# B&R Automation Studio project NAEUL004C00R13L518F00 (part 46)

```iecst
END_ACTION
```

#### Act_OutputConfig.st
```iecst
ACTION Act_OutputConfig:
	// Output: Assign To Global For Independent Package Usage

	g_tyPshrConv := tylocalPshrConv.Out; // Change the Global Naming According to the Physical Hardware Module

END_ACTION
```

#### Cyclic.st
```iecst
(** 2019-03-29 **)
PROGRAM _CYCLIC

	IF bInitialDone = FALSE THEN
		IF g_tyStartUp.bNtSettingsLoadDone = TRUE  THEN
			bInitialDone	:= TRUE;
			Act_Initial;
		END_IF
	ELSE
		Act_InputConfig;
		IF (tylocalPshrConv.In.bPrep = TRUE) AND (tylocalPshrConv.In.bEn = TRUE) AND (tylocalPshrConv.In.bDis = FALSE) THEN
			Act_Link;
			Act_Main;
		ELSE
			IF tylocalPshrConv.Out.eStat <> ConvActIdle THEN
				tylocalPshrConv.Out.eStatus	:= Done;
			ELSE
				tylocalPshrConv.Out.eStatus	:= Idle;
			END_IF
		END_IF
		Act_OutputConfig;
		Act_Alarm;

	END_IF

END_PROGRAM
```

#### Init.st
```iecst
(** 2019-03-25 **)
PROGRAM _INIT

	(* Always Change If Project Change *)

	//Physical Configuration
	diInitTm	:= 0;

	//Pass Address To Global Address For External Use
	//Action, State & Status
	p_PshrConvStat		:= ADR(eStat);
	p_PshrConvStatus	:= ADR(eStatus);
	p_PshrConvStatTxt	:= ADR(sStatTxt);

	//Alarm
	p_PshrConvAlmData	:= ADR(tyAlmData);

	//Output
	p_PshrConvHvBrd						:= ADR(bHvBrd);
	p_PshrConvRejHvBrd					:= ADR(bRejHvBrd);
	p_PshrConvInspHvBrd					:= ADR(bInspHvBrd);
	p_PshrConvGdBrd						:= ADR(bGdBrd);
	p_PshrConvLmtSenActivated			:= ADR(bLmtSenActivated);
	p_PshrConvMtrSigOnOrLToR			:= ADR(bMtrSigOnOrLToR);
	p_PshrConvMtrDirOrRToL				:= ADR(bMtrDirOrRToL);

	p_PshrConvPshrExtCtrl				:= ADR(bPshrExtCtrl);
	p_PshrConvPshrRetCtrl				:= ADR(bPshrRetCtrl);
	p_PshrConvPshrTwoOutputControl		:= ADR(bPshrTwoOutputControl);
	p_PshrConvPshrExtended				:= ADR(bPshrExtended);
	p_PshrConvPshrRetracted				:= ADR(bPshrRetracted);

	p_PshrConvPullerExtCtrl				:= ADR(bPullerExtCtrl);
	p_PshrConvPullerRetCtrl				:= ADR(bPullerRetCtrl);
	p_PshrConvPullerTwoOutputControl	:= ADR(bPullerTwoOutputControl);
	p_PshrConvPullerExtended			:= ADR(bPullerExtended);
	p_PshrConvPullerRetracted			:= ADR(bPullerRetracted);

	p_PshrConvRotRemoteCtrl				:= ADR(bRotRemoteCtrl);
	p_PshrConvRotTwoOutputControl		:= ADR(bRotTwoOutputControl);
	p_PshrConvRotAtRemote				:= ADR(bRotAtRemote);
	p_PshrConvRotAtHome					:= ADR(bRotAtHome);

	p_PshrConvRejectUpCtrl				:= ADR(bRejectUpCtrl);
	p_PshrConvRejectDownCtrl			:= ADR(bRejectDownCtrl);
	p_PshrConvRejectTwoOutputControl	:= ADR(bRejectTwoOutputControl);
	p_PshrConvRejectAtUp				:= ADR(bRejectAtUp);
	p_PshrConvRejectAtDown				:= ADR(bRejectAtDown);
	//ADDED

	p_PshrConvPshrRetAllwTrav			:= ADR(bPshrRetAllwTraverse);

	(* Always Change If Project Change *)

END_PROGRAM
```

### MtrPshr.typ - Change By Project
```iecst
(*2019-06-17*)
(**)
(*Action*)

TYPE
	eMtrPshrAction :
		(
		MtrPshrActIdle,
		MtrPshrActExt,
		MtrPshrActRet,
		MtrPshrActStop,
		MtrPshrActSetExt,
		MtrPshrActRstExt,
		MtrPshrActSetRet,
		MtrPshrActRstRet,
		MtrPshrActSetSpdBit0,
		MtrPshrActRstSpdBit0,
		MtrPshrActSetSpdBit1,
		MtrPshrActRstSpdBit1,
		MtrPshrActSetSpdBit2,
		MtrPshrActRstSpdBit2,
		MtrPshrActSetSigOn,
		MtrPshrActRstSigOn,
		MtrPshrActSetBrake,
		MtrPshrActRstBrake,
		MtrPshrActSetAlmRst,
		MtrPshrActRstAlmRst,
		MtrPshrActSetAll,
		MtrPshrActRstAll
		);
	tyMtrPshr : 	STRUCT
		In : tyMtrPshrIn1;
		Out : tyMtrPshrOut1;
	END_STRUCT;
	tyMtrPshrIn1 : 	STRUCT
		eAct : eConvAction;
		udiRstErr : UDINT;
		bPrep : BOOL;
		bEn : BOOL;
		bDis : BOOL;
		bManual : BOOL;
		bDir : BOOL := FALSE;
		tAlmRstTm : TIME := T#1s;
		tAlmTrigTm : TIME := T#1s;
		tMtrBrkOffDlyTm : TIME := T#500ms;
		tExtTO : TIME := T#20s;
		tRetTO : TIME := T#20s;
		diExtSlowSpd : DINT;
		diRetSlowSpd : DINT;
		diExtNomSpd : {REDUND_UNREPLICABLE} DINT;
		diRetNomSpd : {REDUND_UNREPLICABLE} DINT;
		diExtTorque : DINT;
		diRetTorque : DINT;
		diStartTorque : DINT;
		bExtSen : BOOL;
		bRetSen : BOOL;
		bExtSlowSen : BOOL;
		bRetSlowSen : BOOL;
		bExtSafetySen : BOOL := TRUE;
		bRetSafetySen : BOOL := TRUE;
		bAlarmSig : BOOL;
		bTorqueSig : BOOL;
		bNtParamAutoRcpPrep : BOOL;
		bMcParamAutoRcpDis : BOOL;
		bLinkDISafetyRlySig : BOOL;
		bLinkPshrExtCtrl : BOOL;
		bLinkPshrRetCtrl : BOOL;
		bLinkAlarmSig : BOOL;
		sProgNm : STRING[15];
	END_STRUCT;
	tyMtrPshrOut1 : 	STRUCT
		eStat : eMagConv2ClpAction;
		eStatus : eFBStatus;
		sStatTxt : STRING[200];
		tyAlmData : tyAlmDat;
		bExtended : BOOL;
		bRetracted : BOOL;
		bCW : BOOL;
		bCCW : BOOL;
		bSpdBinBit0 : BOOL;
		bSpdBinBit1 : BOOL;
		bSpdBinBit2 : BOOL;
		bSigOn : BOOL;
		bBrake : BOOL;
		bAlmRst : BOOL;
	END_STRUCT;
END_TYPE
```

### MtrPshr.var - Change By Project
```iecst
VAR
	g_tyMtrPshr : tyMtrPshrOut1;
END_VAR
```

### Program Logical/MtrPshr/MtrPshr (IEC) - 1.00.0 - NtConv v5.00.0 , NtPneu v5.00.0

#### InputRef.var
```iecst
(*2019-03-25*)
(**)
(*General*)
VAR
	p_eAct : REFERENCE TO eMtrPshrAction;
	p_udiRstErr : REFERENCE TO UDINT;
	p_bPrep : REFERENCE TO BOOL;
	p_bEn : REFERENCE TO BOOL;
	p_bDis : REFERENCE TO BOOL;
END_VAR
(**)
(*Configuration*)
VAR
	p_bManual : REFERENCE TO BOOL;
	p_bDir : REFERENCE TO BOOL;
	p_tAlmRstTm : REFERENCE TO TIME;
	p_tAlmTrigTm : REFERENCE TO TIME;
	p_tMtrBrkOffDlyTm : REFERENCE TO TIME;
	p_tExtTO : REFERENCE TO TIME;
	p_tRetTO : REFERENCE TO TIME;
	p_diExtSlowSpd : REFERENCE TO DINT;
	p_diRetSlowSpd : REFERENCE TO DINT;
	p_diExtNomSpd : REFERENCE TO DINT;
	p_diRetNomSpd : REFERENCE TO DINT;
	p_diExtTorque : REFERENCE TO DINT;
	p_diRetTorque : REFERENCE TO DINT;
	p_diStartTorque : REFERENCE TO DINT;
	p_sProgNm : REFERENCE TO STRING[15];
	p_bNtSettingsLoadDone : REFERENCE TO BOOL;
END_VAR
(**)
(*Input*)
VAR
	p_bExtSen : REFERENCE TO BOOL;
	p_bRetSen : REFERENCE TO BOOL;
	p_bExtSlowSen : REFERENCE TO BOOL;
	p_bRetSlowSen : REFERENCE TO BOOL;
	p_bExtSafetySen : REFERENCE TO BOOL;
	p_bRetSafetySen : REFERENCE TO BOOL;
	p_bAlarmSig : REFERENCE TO BOOL;
	p_bTorqueSig : REFERENCE TO BOOL;
	p_bNtParamAutoRcpPrep : REFERENCE TO BOOL;
	p_bMcParamAutoRcpDis : REFERENCE TO BOOL;
END_VAR
```

#### InputRef_Link.var
```iecst
(*2019-04-09*)
(**)
VAR
	p_bLinkOpsRun : REFERENCE TO BOOL;
END_VAR
(**)
VAR
	p_bLinkDISafetyRlySig : REFERENCE TO BOOL;
	p_bLinkPshrExtCtrl : REFERENCE TO BOOL;
	p_bLinkPshrRetCtrl : REFERENCE TO BOOL;
	p_bLinkAlarmSig : REFERENCE TO BOOL;
END_VAR
```

#### Local.var
```iecst
(*2019-06-17*)
VAR
	tylocalMtrPshr : tyMtrPshr;
END_VAR
(**)
(*Local Action, State & Status*)
VAR
	udiStatus : UDINT := 0;
	a_sStatText : ARRAY[0..60] OF STRING[200] := ['Idling','Extending','Retracting','Stopping','Turning On Motor Extend','Turning Off Motor Extend','Turning On Motor Retract','Turning Off Motor Retract','Turning On Speed Binary Bit 0','Turning Off Speed Binary Bit 0','Turning On Speed Binary Bit 1','Turning Off Speed Binary Bit 1','Turning On Speed Binary Bit 2','Turning Off Speed Binary Bit 2','Turning On Signal On','Turning Off Signal On','Turning On Brake','Turning Off Brake','Turning On Alarm Reset','Turning Off Alarm Reset','Turning On All Motor Output','Turning Of All Motor Output',39('')];
END_VAR
(**)
(*Local Alarm*)
VAR
	tyAlmData : tyAlmDat;
END_VAR
(**)
(*Local*)
VAR
	bRstErr : BOOL;
	udiRstErrOld : UDINT;
	bInitDone : BOOL;
	bInitialDone : BOOL;
	eStatOld : eMtrPshrAction := MtrPshrActIdle;
	iAnalogTorque : INT;
	diMtrSpd : DINT;
	bMtrSpdSlw : BOOL;
	fbAlmRstTm : TON := (PT:=T#1s);
	fbAlmTrigTm : TON := (PT:=T#2s);
	fbMtrBrkOffDlyTm : TON;
	fbMtrPshrExtChk : fbPneuExtRetSenExtChk;
	fbMtrPshrRetChk : fbPneuExtRetSenRetChk;
	udiModuleNum : UDINT := 2201;
END_VAR
```

#### Act_Action.st
```iecst
(** 2019-03-25 **)
ACTION Act_Action:

	//Reset Error
	IF (eStatus = Error) AND bRstErr THEN
		p_eAct	:= MtrPshrActIdle;
		eStat	:= MtrPshrActIdle;
	END_IF

	//Set p_eAct
	IF eStatus = Idle OR eStatus = Busy OR eStatus = Done THEN
		eStat	:= p_eAct;
	END_IF

END_ACTION
```

#### Act_Alarm.st
```iecst
(** 2019-03-25 **)
ACTION Act_Alarm:
	//Reset Error
	IF (tylocalMtrPshr.Out.eStatus = Error) AND bRstErr THEN
		tylocalMtrPshr.In.eAct	:= MtrPshrActIdle;
		tylocalMtrPshr.Out.eStat	:= MtrPshrActIdle;
	END_IF

	IF tylocalMtrPshr.In.udiRstErr <> udiRstErrOld THEN
		bRstErr			:= TRUE;
		udiRstErrOld	:= tylocalMtrPshr.In.udiRstErr;
	ELSE
		bRstErr			:= FALSE;
	END_IF
	//Error
	IF EDGEPOS(eStatus = Error) THEN

		tylocalMtrPshr.Out.tyAlmData.udiCode		:= udiStatus;
		tylocalMtrPshr.Out.tyAlmData.eSeverity		:= AlmSeverityError;
		tylocalMtrPshr.Out.tyAlmData.udiRunTime	:= tylocalMtrPshr.Out.tyAlmData.udiRunTime + 1;
		tylocalMtrPshr.Out.tyAlmData.bAlm			:= TRUE;
		tylocalMtrPshr.Out.tyAlmData.udiModuleNum  := udiModuleNum;
		g_tyAlmProgNm.sMtrPshrProgNm		    := tylocalMtrPshr.In.sProgNm;

		tylocalMtrPshr.Out.sStatTxt	:= tylocalMtrPshr.Out.tyAlmData.sAlmMsg;

	ELSIF bRstErr AND (tyAlmData.udiCode <> 0) THEN

		tylocalMtrPshr.Out.tyAlmData.udiCode	:= 0;
		tylocalMtrPshr.Out.tyAlmData.eSeverity	:= AlmSeverityNA;
		tylocalMtrPshr.Out.tyAlmData.bAlm			:= FALSE;
		tylocalMtrPshr.Out.sStatTxt	:= a_sStatText[tylocalMtrPshr.Out.eStat];

	END_IF

END_ACTION
```

#### Act_Background.st
```iecst
(** 2019-01-18 **)
ACTION Act_Background:

	//background
	IF tylocalMtrPshr.In.bExtSen = FALSE THEN
		tylocalMtrPshr.Out.bExtended	:= FALSE;
	END_IF

	IF tylocalMtrPshr.In.bRetSen = FALSE THEN
		tylocalMtrPshr.Out.bRetracted	:= FALSE;
	END_IF

	//Torque Minimum Value
	IF iAnalogTorque < 1500 THEN
		iAnalogTorque	:= 1500;
	END_IF

	//Abnormal Movement
	IF tylocalMtrPshr.Out.eStatus <> Error THEN

		fbAlmTrigTm(IN := NOT tylocalMtrPshr.In.bAlarmSig);

		IF fbAlmTrigTm.Q = TRUE THEN
			tylocalMtrPshr.Out.eStatus		:= Error;
			udiStatus	:= 10006;	//Motorized Pusher Alarm Occur

			tylocalMtrPshr.Out.bCW			:= FALSE;
			tylocalMtrPshr.Out.bCCW		:= FALSE;
			tylocalMtrPshr.Out.bSpdBinBit0	:= FALSE;
			tylocalMtrPshr.Out.bSpdBinBit1	:= FALSE;
			tylocalMtrPshr.Out.bSpdBinBit2	:= FALSE;
			tylocalMtrPshr.Out.bSigOn		:= FALSE;
			tylocalMtrPshr.Out.bBrake		:= FALSE;
			tylocalMtrPshr.Out.bAlmRst		:= FALSE;

			tylocalMtrPshr.In.eAct	:= MtrPshrActIdle;
			tylocalMtrPshr.Out.eStat	:= MtrPshrActIdle;
		END_IF

	END_IF

	//Reset Error
	IF (tylocalMtrPshr.Out.eStatus = Error) AND bRstErr THEN
		IF tylocalMtrPshr.In.bAlarmSig = FALSE THEN
			tylocalMtrPshr.Out.bAlmRst			:= TRUE;
			fbAlmRstTm.IN	:= TRUE;
			fbAlmTrigTm(IN := FALSE);
		END_IF
	END_IF

	fbAlmRstTm;

	IF fbAlmRstTm.Q = TRUE THEN
		tylocalMtrPshr.Out.bAlmRst		:= FALSE;
		tylocalMtrPshr.Out.eStatus		:= Idle;
		udiStatus	:= 0;

		fbAlmRstTm.IN	:= FALSE;
	END_IF
END_ACTION
```

#### Act_InitGlobal.st
```iecst
(** 2019-04-09 **)
ACTION Act_InitGlobal:

	(* Always Change If Project Change *)

	//Pass Data To Link
	p_bLinkOpsRun ACCESS p_OpsRun;

	p_bLinkDISafetyRlySig ACCESS p_DISafetyRlySig;
	p_bLinkPshrExtCtrl ACCESS p_PshrConvPshrExtCtrl;
	p_bLinkPshrRetCtrl ACCESS p_PshrConvPshrRetCtrl;
	p_bLinkAlarmSig ACCESS p_DIMtrPshrAlmSig;

	//Pass Data To Internal Use
	p_udiRstErr ACCESS p_RstErrReset;
	p_bPrep ACCESS p_NtParamProjMotorizedPusherPrep;
	p_bManual ACCESS p_UIMnlMod;
	p_bDir ACCESS p_NtParamMtrPshrDir;
	p_tExtTO ACCESS p_NtParamMtrPshrExtTO;
	p_tRetTO ACCESS p_NtParamMtrPshrRetTO;
	p_diExtSlowSpd ACCESS p_NtParamMtrPshrExtSlowSpd;
	p_diRetSlowSpd ACCESS p_NtParamMtrPshrRetSlowSpd;
	p_diRetNomSpd ACCESS p_NtParamMtrPshrRetNomSpd;
	p_diRetTorque ACCESS p_NtParamMtrPshrRetTorq;
	p_diStartTorque ACCESS p_NtParamMtrPshrStartTorq;
	p_sProgNm ACCESS p_NtParamMtrPshrProgNm;
	p_bNtSettingsLoadDone ACCESS p_StartupNtSettingsLoadDone;

	p_bExtSen ACCESS p_DIPusherExtRS;
	p_bRetSen ACCESS p_DIPusherRetRS;
	p_bExtSlowSen ACCESS p_DIPusherExtSlwSen;
	p_bRetSlowSen ACCESS p_DIPusherRetSlwSen;
//	p_bAlarmSig ACCESS p_DIMtrPshrAlmSig;
	p_bTorqueSig ACCESS p_DIMtrPshrTorqueSig;

	p_bNtParamAutoRcpPrep ACCESS p_NtParamAutoRcpPrep ;
	p_bMcParamAutoRcpDis  ACCESS p_McParamAutoRcpDisable;
	(* Always Change If Project Change *)

END_ACTION
```

#### Act_Initial.st
```iecst
(** 2019-03-22 **)
ACTION Act_Initial:

	//Initial
	tylocalMtrPshr.Out.sStatTxt	:=  a_sStatText[eStat];

	fbAlmRstTm(IN := FALSE);
	fbAlmTrigTm(IN := FALSE);
	fbMtrBrkOffDlyTm(IN :=FALSE);
	fbMtrPshrExtChk(bEn	:=FALSE);
	fbMtrPshrRetChk(bEn	:=FALSE);

END_ACTION
```

#### Act_InitLocal.st
```iecst
(** 2019-03-25 **)
ACTION Act_InitLocal:

	//Input Reference Link To Local Variable
	p_eAct ACCESS ADR(eAct);
	p_udiRstErr ACCESS ADR(udiRstErr);
	p_bPrep ACCESS ADR(bPrep);
	p_bEn ACCESS ADR(bEn);
	p_bDis ACCESS ADR(bDis);

	p_bManual ACCESS ADR(bManual);
	p_bDir ACCESS ADR(bDir);
	p_tAlmRstTm ACCESS ADR(tAlmRstTm);
	p_tAlmTrigTm ACCESS ADR(tAlmTrigTm);
	p_tMtrBrkOffDlyTm ACCESS ADR(tMtrBrkOffDlyTm);
	p_tExtTO ACCESS ADR(tExtTO);
	p_tRetTO ACCESS ADR(tRetTO);
	p_diExtSlowSpd ACCESS ADR(diExtSlowSpd);
	p_diRetSlowSpd ACCESS ADR(diRetSlowSpd);
	p_diExtNomSpd ACCESS ADR(diExtNomSpd);
	p_diRetNomSpd ACCESS ADR(diRetNomSpd);
	p_diExtTorque ACCESS ADR(diExtTorque);
	p_diRetTorque ACCESS ADR(diRetTorque);
	p_diStartTorque ACCESS ADR(diStartTorque);
	p_sProgNm ACCESS ADR(sProgNm);
	p_bNtSettingsLoadDone ACCESS ADR(bNtSettingsLoadDone);

	p_bExtSen ACCESS ADR(bExtSen);
	p_bRetSen ACCESS ADR(bRetSen);
	p_bExtSlowSen ACCESS ADR(bExtSlowSen);
	p_bRetSlowSen ACCESS ADR(bRetSlowSen);
	p_bExtSafetySen ACCESS ADR(bExtSafetySen);
	p_bRetSafetySen ACCESS ADR(bRetSafetySen);
	p_bAlarmSig ACCESS ADR(bAlarmSig);
	p_bTorqueSig ACCESS ADR(bTorqueSig);

END_ACTION
```

#### Act_InputConfig.st
```iecst
(** 2019-04-09 **)
ACTION Act_InputConfig:

	(* Always Change If Project Change *)

	//Pass Data To Link

	tylocalMtrPshr.In.bLinkDISafetyRlySig := g_tyDISafetyRlySig;
	tylocalMtrPshr.In.bLinkPshrExtCtrl := g_tyPshrConvPshrExtCtrl;
	tylocalMtrPshr.In.bLinkPshrRetCtrl := g_tyPshrConvPshrRetCtrl;
	tylocalMtrPshr.In.bLinkAlarmSig := g_tyDIMtrPshrAlmSig;

	//Pass Data To Internal Use
	tylocalMtrPshr.In.udiRstErr := g_tyRstErrReset;
	tylocalMtrPshr.In.bPrep := g_tyNtParamProjMotorizedPusherPrep;
	tylocalMtrPshr.In.bManual := g_tyUIMnlMod;
	tylocalMtrPshr.In.bDir := g_tyNtParamMtrPshrDir;
	tylocalMtrPshr.In.tExtTO := g_tyNtParamMtrPshrExtTO;
	tylocalMtrPshr.In.tRetTO := g_tyNtParamMtrPshrRetTO;
	tylocalMtrPshr.In.diExtSlowSpd := g_tyNtParamMtrPshrExtSlowSpd;
	tylocalMtrPshr.In.diRetSlowSpd := g_tyNtParamMtrPshrRetSlowSpd;
	tylocalMtrPshr.In.diRetNomSpd := g_tyNtParamMtrPshrRetNomSpd;
	tylocalMtrPshr.In.diRetTorque := g_tyNtParamMtrPshrRetTorq;
	tylocalMtrPshr.In.diStartTorque := g_tyNtParamMtrPshrStartTorq;
	tylocalMtrPshr.In.sProgNm := g_tyNtParamCurr.sMtrPshrProgNm;

	tylocalMtrPshr.In.bExtSen := g_tyDIPusherExtRS;
	tylocalMtrPshr.In.bRetSen := g_tyDIPusherRetRS;
	tylocalMtrPshr.In.bExtSlowSen := g_tyDIPusherExtSlwSen;
	tylocalMtrPshr.In.bRetSlowSen := g_tyDIPusherRetSlwSen;
//	tylocalMtrPshr.In.bAlarmSig := g_tyDIMtrPshrAlmSig;
	tylocalMtrPshr.In.bTorqueSig := g_tyDIMtrPshrTorqueSig;

	tylocalMtrPshr.In.bNtParamAutoRcpPrep := g_tyNtParamAutoRcpPrep ;
	tylocalMtrPshr.In.bMcParamAutoRcpDis  := g_tyMcParamAutoRcpDisable;
	(* Always Change If Project Change *)

	IF g_tyOps.bRun THEN

		IF (tylocalMtrPshr.Out.eStatus <> Busy AND tylocalMtrPshr.Out.eStatus <> Idle)OR (tylocalMtrPshr.In.bLinkPshrExtCtrl = FALSE AND tylocalMtrPshr.In.bLinkPshrRetCtrl = FALSE)  THEN
			tylocalMtrPshr.In.eAct := MtrPshrActIdle;
		ELSIF tylocalMtrPshr.In.bLinkPshrExtCtrl AND tylocalMtrPshr.In.bLinkPshrRetCtrl = FALSE
			AND tylocalMtrPshr.In.bExtSen = FALSE
			THEN
			tylocalMtrPshr.In.eAct := MtrPshrActExt;

		ELSIF tylocalMtrPshr.In.bLinkPshrExtCtrl = FALSE AND tylocalMtrPshr.In.bLinkPshrRetCtrl
			AND tylocalMtrPshr.In.bRetSen = FALSE
			THEN
			tylocalMtrPshr.In.eAct := MtrPshrActRet;
		END_IF

	ELSIF tylocalMtrPshr.In.bManual = TRUE THEN

		IF (tylocalMtrPshr.Out.eStatus <> Busy AND tylocalMtrPshr.Out.eStatus <> Idle)OR (tylocalMtrPshr.In.bLinkPshrExtCtrl = FALSE AND tylocalMtrPshr.In.bLinkPshrRetCtrl = FALSE)  THEN
			tylocalMtrPshr.In.eAct := MtrPshrActIdle;
		ELSIF tylocalMtrPshr.In.bLinkPshrExtCtrl AND tylocalMtrPshr.In.bLinkPshrRetCtrl = FALSE
			AND tylocalMtrPshr.In.bExtSen = FALSE
			THEN
			tylocalMtrPshr.In.eAct := MtrPshrActExt;

		ELSIF tylocalMtrPshr.In.bLinkPshrExtCtrl = FALSE AND tylocalMtrPshr.In.bLinkPshrRetCtrl
			AND tylocalMtrPshr.In.bRetSen = FALSE
			THEN
			tylocalMtrPshr.In.eAct := MtrPshrActRet;
		END_IF

	ELSE
		tylocalMtrPshr.In.eAct := MtrPshrActIdle;
	END_IF
END_ACTION
```

#### Act_Link.st
```iecst
(** 2019-03-29 **)
ACTION Act_Link:

	IF tylocalMtrPshr.In.bLinkDISafetyRlySig = FALSE THEN
		tylocalMtrPshr.Out.bExtended	:= FALSE;
		tylocalMtrPshr.Out.bRetracted	:= FALSE;
	END_IF

	IF tylocalMtrPshr.In.bManual = TRUE THEN
		tylocalMtrPshr.In.diExtNomSpd ACCESS ADR(g_tyUIMnlMtrPshrExtSpd);
		tylocalMtrPshr.In.diExtTorque ACCESS ADR(g_tyUIMnlMtrPshrExtTorq);
	ELSE
		IF tylocalMtrPshr.In.bNtParamAutoRcpPrep AND NOT(tylocalMtrPshr.In.bMcParamAutoRcpDis) THEN
			tylocalMtrPshr.In.diExtNomSpd ACCESS g_tyProdRcpCurrRcp0MtrPshrExtSpd;
			tylocalMtrPshr.In.diExtTorque ACCESS g_tyProdRcpCurrRcp0MtrPshrExtTorq;
		ELSE
			tylocalMtrPshr.In.diExtNomSpd ACCESS  g_tyProdRcpCurrRcp1MtrPshrExtSpd;
			tylocalMtrPshr.In.diExtTorque ACCESS g_tyProdRcpCurrRcp1MtrPshrExtTorq;
		END_IF
	END_IF

	IF tylocalMtrPshr.In.bLinkDISafetyRlySig = TRUE THEN
		tylocalMtrPshr.In.bAlarmSig := tylocalMtrPshr.In.bLinkAlarmSig;
	ELSE
		tylocalMtrPshr.In.bAlarmSig := TRUE;
	END_IF

END_ACTION
```

#### Act_LinkAction.st
```iecst
(** 2019-04-09 **)
ACTION Act_LinkAction:

	IF p_bLinkOpsRun = TRUE THEN
		//	p_eAct ACCESS p_OpsTravULMtrPshrAct;
		IF p_bLinkPshrExtCtrl AND p_bLinkPshrRetCtrl = FALSE
			AND p_bExtSen = FALSE
			THEN
				p_eAct := MtrPshrActExt;

		ELSIF p_bLinkPshrExtCtrl = FALSE AND p_bLinkPshrRetCtrl
			AND p_bRetSen = FALSE
			THEN
				p_eAct := MtrPshrActRet;

		ELSE
				p_eAct := MtrPshrActIdle;
		END_IF

	ELSIF p_bManual = TRUE THEN
//		IF p_UIMtrPshrAct = MtrPshrActStop THEN
//			p_eAct := MtrPshrActStop;
//		ELSE
			IF p_bLinkPshrExtCtrl AND p_bLinkPshrRetCtrl = FALSE
			AND p_bExtSen = FALSE
				THEN
				p_eAct := MtrPshrActExt;

			ELSIF p_bLinkPshrExtCtrl = FALSE AND p_bLinkPshrRetCtrl
				AND p_bRetSen = FALSE
				THEN
				p_eAct := MtrPshrActRet;

			ELSE
				p_eAct := MtrPshrActIdle;
			END_IF
//		END_IF

	ELSE
			p_eAct := MtrPshrActIdle;
	END_IF

END_ACTION
```

#### Act_LinkEn.st
```iecst
(** 2019-01-11 **)
ACTION Act_LinkEn:

	//Link bPrep, bEn & bDis
	//p_bEn	:= FALSE;

END_ACTION
```

#### Act_Main.st
```iecst
(** 2019-06-17 **)
ACTION Act_Main:

	fbAlmRstTm.PT				:= tylocalMtrPshr.In.tAlmRstTm;
	fbAlmTrigTm.PT				:= tylocalMtrPshr.In.tAlmTrigTm;
	fbMtrBrkOffDlyTm.PT			:= tylocalMtrPshr.In.tMtrBrkOffDlyTm;
	fbMtrPshrExtChk.tTimeOut	:= tylocalMtrPshr.In.tExtTO;
	fbMtrPshrRetChk.tTimeOut	:= tylocalMtrPshr.In.tRetTO;
	//Set tylocalMtrPshr.In.eAct
	IF tylocalMtrPshr.Out.eStatus = Idle OR tylocalMtrPshr.Out.eStatus = Busy OR tylocalMtrPshr.Out.eStatus = Done THEN
		tylocalMtrPshr.Out.eStat	:= tylocalMtrPshr.In.eAct;
	END_IF

	IF eStatOld <> tylocalMtrPshr.Out.eStat THEN
		bMtrSpdSlw	:= FALSE;

		fbMtrBrkOffDlyTm(IN := FALSE);
		fbMtrPshrExtChk(bEn := FALSE);
		fbMtrPshrRetChk(bEn := FALSE);

		IF eStatOld <> MtrPshrActIdle
			AND eStatOld <> MtrPshrActSetExt
			AND eStatOld <> MtrPshrActRstExt
			AND eStatOld <> MtrPshrActSetRet
			AND eStatOld <> MtrPshrActRstRet
			AND eStatOld <> MtrPshrActSetSpdBit0
			AND eStatOld <> MtrPshrActRstSpdBit0
			AND eStatOld <> MtrPshrActSetSpdBit1
			AND eStatOld <> MtrPshrActRstSpdBit1
			AND eStatOld <> MtrPshrActSetSpdBit2
			AND eStatOld <> MtrPshrActRstSpdBit2
			AND eStatOld <> MtrPshrActSetSigOn
			AND eStatOld <> MtrPshrActRstSigOn
			AND eStatOld <> MtrPshrActSetBrake
			AND eStatOld <> MtrPshrActRstBrake
			AND eStatOld <> MtrPshrActSetAlmRst
			AND eStatOld <> MtrPshrActRstAlmRst
			AND eStatOld <> MtrPshrActSetAll
			AND eStatOld <> MtrPshrActRstAll THEN

			tylocalMtrPshr.Out.bCW			:= FALSE;
			tylocalMtrPshr.Out.bCCW		:= FALSE;
			tylocalMtrPshr.Out.bSpdBinBit0	:= FALSE;
			tylocalMtrPshr.Out.bSpdBinBit1	:= FALSE;
			tylocalMtrPshr.Out.bSpdBinBit2	:= FALSE;
			tylocalMtrPshr.Out.bSigOn		:= FALSE;
			tylocalMtrPshr.Out.bBrake		:= FALSE;
			tylocalMtrPshr.Out.bAlmRst		:= FALSE;

		END_IF

		sStatTxt	:= a_sStatText[tylocalMtrPshr.Out.eStat];

		eStatOld	:= tylocalMtrPshr.Out.eStat;

		tylocalMtrPshr.Out.eStatus		:= Busy;
	END_IF

	//Main
	CASE tylocalMtrPshr.Out.eStat OF

		MtrPshrActIdle:
			IF EDGENEG(tylocalMtrPshr.In.bManual) THEN
				tylocalMtrPshr.Out.bCW			:= FALSE;
				tylocalMtrPshr.Out.bCCW		:= FALSE;
				tylocalMtrPshr.Out.bSpdBinBit0	:= FALSE;
				tylocalMtrPshr.Out.bSpdBinBit1	:= FALSE;
				tylocalMtrPshr.Out.bSpdBinBit2	:= FALSE;
				tylocalMtrPshr.Out.bSigOn		:= FALSE;
				tylocalMtrPshr.Out.bBrake		:= FALSE;
				tylocalMtrPshr.Out.bAlmRst		:= FALSE;
			END_IF

			tylocalMtrPshr.Out.eStatus	:= Idle;

		MtrPshrActExt:
			IF tylocalMtrPshr.Out.eStatus = Idle OR tylocalMtrPshr.Out.eStatus = Busy THEN
				tylocalMtrPshr.Out.eStatus	:= Busy;

				//Motor Torque
				IF (tylocalMtrPshr.In.bRetSen OR tylocalMtrPshr.In.bRetSlowSen) THEN// OR  NOT(bMtrSpdSlw) THEN
					iAnalogTorque	:= ((DINT_TO_INT(tylocalMtrPshr.In.diStartTorque) * 16383) / 100); //5V at 16383 for maximum Torque
				ELSE //IF bMtrSpdSlw THEN
					iAnalogTorque	:= ((DINT_TO_INT(tylocalMtrPshr.In.diExtTorque) * 16383) / 100);
				END_IF

				IF iAnalogTorque < 1500 THEN
					iAnalogTorque	:= 1500;
				END_IF

				//Motor Speed
				IF tylocalMtrPshr.In.bExtSlowSen = TRUE OR tylocalMtrPshr.In.bTorqueSig = TRUE THEN
					bMtrSpdSlw	:= TRUE;
				END_IF

				IF bMtrSpdSlw = TRUE THEN
					diMtrSpd	:= tylocalMtrPshr.In.diExtSlowSpd;
				ELSE
					diMtrSpd	:= tylocalMtrPshr.In.diExtNomSpd;
				END_IF

				CASE diMtrSpd OF
					1:
						tylocalMtrPshr.Out.bSpdBinBit0	:= FALSE;
						tylocalMtrPshr.Out.bSpdBinBit1	:= FALSE;
						tylocalMtrPshr.Out.bSpdBinBit2	:= FALSE;
					2:
						tylocalMtrPshr.Out.bSpdBinBit0	:= TRUE;
						tylocalMtrPshr.Out.bSpdBinBit1	:= FALSE;
						tylocalMtrPshr.Out.bSpdBinBit2	:= FALSE;
					3:
						tylocalMtrPshr.Out.bSpdBinBit0	:= FALSE;
						tylocalMtrPshr.Out.bSpdBinBit1	:= TRUE;
						tylocalMtrPshr.Out.bSpdBinBit2	:= FALSE;
					4:
						tylocalMtrPshr.Out.bSpdBinBit0	:= TRUE;
						tylocalMtrPshr.Out.bSpdBinBit1	:= TRUE;
						tylocalMtrPshr.Out.bSpdBinBit2	:= FALSE;
					5:
						tylocalMtrPshr.Out.bSpdBinBit0	:= FALSE;
						tylocalMtrPshr.Out.bSpdBinBit1	:= FALSE;
						tylocalMtrPshr.Out.bSpdBinBit2	:= TRUE;
					6:
						tylocalMtrPshr.Out.bSpdBinBit0	:= TRUE;
						tylocalMtrPshr.Out.bSpdBinBit1	:= FALSE;
						tylocalMtrPshr.Out.bSpdBinBit2	:= TRUE;
					7:
						tylocalMtrPshr.Out.bSpdBinBit0	:= FALSE;
						tylocalMtrPshr.Out.bSpdBinBit1	:= TRUE;
						tylocalMtrPshr.Out.bSpdBinBit2	:= TRUE;
					8:
						tylocalMtrPshr.Out.bSpdBinBit0	:= TRUE;
						tylocalMtrPshr.Out.bSpdBinBit1	:= TRUE;
						tylocalMtrPshr.Out.bSpdBinBit2	:= TRUE;
				END_CASE

				//Motor On
				tylocalMtrPshr.Out.bSigOn	:= FALSE;
				tylocalMtrPshr.Out.bBrake	:= TRUE;

				IF tylocalMtrPshr.In.bDir = TRUE THEN
					tylocalMtrPshr.Out.bCW		:= TRUE;
				ELSE
					tylocalMtrPshr.Out.bCCW	:= TRUE;
				END_IF

				//Checking Extend
				fbMtrPshrExtChk.bExtSen		:= tylocalMtrPshr.In.bExtSen;
				fbMtrPshrExtChk.bRetSen		:= tylocalMtrPshr.In.bRetSen;
				fbMtrPshrExtChk.bExtSafety	:= tylocalMtrPshr.In.bExtSafetySen;

				fbMtrPshrExtChk(bEn := TRUE);

				IF fbMtrPshrExtChk.udiStatus = 0 THEN

					tylocalMtrPshr.Out.bSigOn	:= TRUE;
					tylocalMtrPshr.Out.bBrake	:= FALSE;
					tylocalMtrPshr.Out.bCW		:= FALSE;
					tylocalMtrPshr.Out.bCCW	:= FALSE;

					fbMtrBrkOffDlyTm(IN := TRUE);

					IF fbMtrBrkOffDlyTm.Q = TRUE THEN
						fbMtrBrkOffDlyTm(IN := FALSE);

						tylocalMtrPshr.Out.bCW			:= FALSE;
						tylocalMtrPshr.Out.bCCW		:= FALSE;
						tylocalMtrPshr.Out.bSpdBinBit0	:= FALSE;
						tylocalMtrPshr.Out.bSpdBinBit1	:= FALSE;
						tylocalMtrPshr.Out.bSpdBinBit2	:= FALSE;
						tylocalMtrPshr.Out.bSigOn		:= FALSE;
						tylocalMtrPshr.Out.bBrake		:= FALSE;

						tylocalMtrPshr.Out.bExtended	:= TRUE;
						tylocalMtrPshr.Out.eStatus		:= Done;
					END_IF

				ELSIF fbMtrPshrExtChk.udiStatus < 65534 THEN

					tylocalMtrPshr.Out.bCW			:= FALSE;
					tylocalMtrPshr.Out.bCCW		:= FALSE;
					tylocalMtrPshr.Out.bSpdBinBit0	:= FALSE;
					tylocalMtrPshr.Out.bSpdBinBit1	:= FALSE;
					tylocalMtrPshr.Out.bSpdBinBit2	:= FALSE;
					tylocalMtrPshr.Out.bSigOn		:= TRUE;
					tylocalMtrPshr.Out.bBrake		:= FALSE;

					tylocalMtrPshr.Out.bExtended	:= FALSE;
					tylocalMtrPshr.Out.eStatus		:= Error;

					IF fbMtrPshrExtChk.udiStatus = 1506 THEN
						udiStatus	:= 10000;	//Pusher Retract Sensor Off Time Out In Extend Check While Pusher Extend
					ELSIF fbMtrPshrExtChk.udiStatus = 1503 THEN
						udiStatus	:= 10001;	//Pusher Extend Sensor On Time Out In Extend Check While Pusher Extend
					ELSIF fbMtrPshrExtChk.udiStatus = 1507 THEN
						udiStatus	:= 10002;	//Pusher Extend Safety Sensor Error In Extend Check While Pusher Extend
					ELSE
						udiStatus	:= fbMtrPshrExtChk.udiStatus;
					END_IF

				END_IF

			END_IF

		MtrPshrActRet:
			IF tylocalMtrPshr.Out.eStatus = Idle OR tylocalMtrPshr.Out.eStatus = Busy THEN
				tylocalMtrPshr.Out.eStatus	:= Busy;

				//Motor Torque
				IF (tylocalMtrPshr.In.bExtSen OR tylocalMtrPshr.In.bExtSlowSen) THEN //OR NOT(bMtrSpdSlw) THEN
					iAnalogTorque	:= ((DINT_TO_INT(tylocalMtrPshr.In.diStartTorque) * 16383) / 100); //32767 ==10V ,10000 == 3v
				ELSE // bMtrSpdSlw THEN
					iAnalogTorque	:= ((DINT_TO_INT(tylocalMtrPshr.In.diRetTorque) * 16383) / 100);
				END_IF

				IF iAnalogTorque < 1500 THEN
					iAnalogTorque	:= 1500;
				END_IF

				//Motor Speed
				IF tylocalMtrPshr.In.bRetSlowSen = TRUE THEN
					bMtrSpdSlw	:= TRUE;
				END_IF

				IF bMtrSpdSlw = TRUE THEN
					diMtrSpd	:= tylocalMtrPshr.In.diRetSlowSpd;
				ELSE
					diMtrSpd	:= tylocalMtrPshr.In.diRetNomSpd;
				END_IF

				CASE diMtrSpd OF
					1:
						tylocalMtrPshr.Out.bSpdBinBit0	:= FALSE;
						tylocalMtrPshr.Out.bSpdBinBit1	:= FALSE;
						tylocalMtrPshr.Out.bSpdBinBit2	:= FALSE;
					2:
						tylocalMtrPshr.Out.bSpdBinBit0	:= TRUE;
						tylocalMtrPshr.Out.bSpdBinBit1	:= FALSE;
						tylocalMtrPshr.Out.bSpdBinBit2	:= FALSE;
					3:
						tylocalMtrPshr.Out.bSpdBinBit0	:= FALSE;
						tylocalMtrPshr.Out.bSpdBinBit1	:= TRUE;
						tylocalMtrPshr.Out.bSpdBinBit2	:= FALSE;
					4:
						tylocalMtrPshr.Out.bSpdBinBit0	:= TRUE;
						tylocalMtrPshr.Out.bSpdBinBit1	:= TRUE;
						tylocalMtrPshr.Out.bSpdBinBit2	:= FALSE;
					5:
						tylocalMtrPshr.Out.bSpdBinBit0	:= FALSE;
						tylocalMtrPshr.Out.bSpdBinBit1	:= FALSE;
						tylocalMtrPshr.Out.bSpdBinBit2	:= TRUE;
					6:
						tylocalMtrPshr.Out.bSpdBinBit0	:= TRUE;
						tylocalMtrPshr.Out.bSpdBinBit1	:= FALSE;
						tylocalMtrPshr.Out.bSpdBinBit2	:= TRUE;
					7:
						tylocalMtrPshr.Out.bSpdBinBit0	:= FALSE;
						tylocalMtrPshr.Out.bSpdBinBit1	:= TRUE;
						tylocalMtrPshr.Out.bSpdBinBit2	:= TRUE;
					8:
						tylocalMtrPshr.Out.bSpdBinBit0	:= TRUE;
						tylocalMtrPshr.Out.bSpdBinBit1	:= TRUE;
						tylocalMtrPshr.Out.bSpdBinBit2	:= TRUE;
				END_CASE

				//Motor On
				tylocalMtrPshr.Out.bSigOn	:= FALSE;
				tylocalMtrPshr.Out.bBrake	:= TRUE;

				IF tylocalMtrPshr.In.bDir = TRUE THEN
					tylocalMtrPshr.Out.bCCW	:= TRUE;
				ELSE
					tylocalMtrPshr.Out.bCW		:= TRUE;
				END_IF

				//Checking Retract
				fbMtrPshrRetChk.bExtSen		:= tylocalMtrPshr.In.bExtSen;
				fbMtrPshrRetChk.bRetSen		:= tylocalMtrPshr.In.bRetSen;
				fbMtrPshrRetChk.bRetSafety	:= tylocalMtrPshr.In.bRetSafetySen;

				fbMtrPshrRetChk(bEn := TRUE);

				IF fbMtrPshrRetChk.udiStatus = 0 THEN

					tylocalMtrPshr.Out.bSigOn	:= TRUE;
					tylocalMtrPshr.Out.bBrake	:= FALSE;
					tylocalMtrPshr.Out.bCW		:= FALSE;
					tylocalMtrPshr.Out.bCCW	:= FALSE;

					fbMtrBrkOffDlyTm(IN := TRUE);

					IF fbMtrBrkOffDlyTm.Q = TRUE THEN
						fbMtrBrkOffDlyTm(IN := FALSE);

						tylocalMtrPshr.Out.bCW			:= FALSE;
						tylocalMtrPshr.Out.bCCW		:= FALSE;
						tylocalMtrPshr.Out.bSpdBinBit0	:= FALSE;
						tylocalMtrPshr.Out.bSpdBinBit1	:= FALSE;
						tylocalMtrPshr.Out.bSpdBinBit2	:= FALSE;
						tylocalMtrPshr.Out.bSigOn		:= FALSE;
						tylocalMtrPshr.Out.bBrake		:= FALSE;

						tylocalMtrPshr.Out.bRetracted	:= TRUE;
						tylocalMtrPshr.Out.eStatus		:= Done;
					END_IF

				ELSIF fbMtrPshrRetChk.udiStatus < 65534 THEN

					tylocalMtrPshr.Out.bCW			:= FALSE;
					tylocalMtrPshr.Out.bCCW		:= FALSE;
					tylocalMtrPshr.Out.bSpdBinBit0	:= FALSE;
					tylocalMtrPshr.Out.bSpdBinBit1	:= FALSE;
					tylocalMtrPshr.Out.bSpdBinBit2	:= FALSE;
					tylocalMtrPshr.Out.bSigOn		:= TRUE;
					tylocalMtrPshr.Out.bBrake		:= FALSE;

					tylocalMtrPshr.Out.bRetracted	:= FALSE;
					tylocalMtrPshr.Out.eStatus		:= Error;

					IF fbMtrPshrRetChk.udiStatus = 1504 THEN
						udiStatus	:= 10003;	//Pusher Extend Sensor Off Time Out In Retract Check While Pusher Retract
					ELSIF fbMtrPshrRetChk.udiStatus = 1505 THEN
						udiStatus	:= 10004;	//Pusher Retract Sensor On Time Out In Retract Check While Pusher Retract
					ELSIF fbMtrPshrRetChk.udiStatus = 1508 THEN
						udiStatus	:= 10005;	//Pusher Retract Safety Sensor Error In Retract Check While Pusher Retract
					ELSE
						udiStatus	:= fbMtrPshrRetChk.udiStatus;
					END_IF

				END_IF

			END_IF

		MtrPshrActStop:
			IF tylocalMtrPshr.Out.eStatus = Idle OR tylocalMtrPshr.Out.eStatus = Busy THEN

				tylocalMtrPshr.Out.bCW			:= FALSE;
				tylocalMtrPshr.Out.bCCW		:= FALSE;
				tylocalMtrPshr.Out.bSpdBinBit0	:= FALSE;
				tylocalMtrPshr.Out.bSpdBinBit1	:= FALSE;
				tylocalMtrPshr.Out.bSpdBinBit2	:= FALSE;
				tylocalMtrPshr.Out.bSigOn		:= TRUE;
				tylocalMtrPshr.Out.bBrake		:= FALSE;

				tylocalMtrPshr.Out.eStatus		:= Done;

			END_IF

		MtrPshrActSetExt:
			IF tylocalMtrPshr.Out.eStatus = Idle OR tylocalMtrPshr.Out.eStatus = Busy THEN

				IF tylocalMtrPshr.In.bDir = TRUE THEN
					tylocalMtrPshr.Out.bCW		:= TRUE;
				ELSE
					tylocalMtrPshr.Out.bCCW	:= TRUE;
				END_IF

				tylocalMtrPshr.Out.eStatus		:= Done;

			END_IF

		MtrPshrActRstExt:
			IF tylocalMtrPshr.Out.eStatus = Idle OR tylocalMtrPshr.Out.eStatus = Busy THEN

				IF tylocalMtrPshr.In.bDir = TRUE THEN
					tylocalMtrPshr.Out.bCW		:= FALSE;
				ELSE
					tylocalMtrPshr.Out.bCCW	:= FALSE;
				END_IF

				tylocalMtrPshr.Out.eStatus		:= Done;

			END_IF

		MtrPshrActSetRet:
			IF tylocalMtrPshr.Out.eStatus = Idle OR tylocalMtrPshr.Out.eStatus = Busy THEN

				IF tylocalMtrPshr.In.bDir = TRUE THEN
					tylocalMtrPshr.Out.bCCW	:= TRUE;
				ELSE
					tylocalMtrPshr.Out.bCW		:= TRUE;
				END_IF

				tylocalMtrPshr.Out.eStatus		:= Done;

			END_IF

		MtrPshrActRstRet:
			IF tylocalMtrPshr.Out.eStatus = Idle OR tylocalMtrPshr.Out.eStatus = Busy THEN

				IF tylocalMtrPshr.In.bDir = TRUE THEN
					tylocalMtrPshr.Out.bCCW	:= FALSE;
				ELSE
					tylocalMtrPshr.Out.bCW		:= FALSE;
				END_IF

				tylocalMtrPshr.Out.eStatus		:= Done;

			END_IF

		MtrPshrActSetSpdBit0:
			IF tylocalMtrPshr.Out.eStatus = Idle OR tylocalMtrPshr.Out.eStatus = Busy THEN

				tylocalMtrPshr.Out.bSpdBinBit0	:= TRUE;

				tylocalMtrPshr.Out.eStatus		:= Done;

			END_IF

		MtrPshrActRstSpdBit0:
			IF tylocalMtrPshr.Out.eStatus = Idle OR tylocalMtrPshr.Out.eStatus = Busy THEN

				tylocalMtrPshr.Out.bSpdBinBit0	:= FALSE;

				tylocalMtrPshr.Out.eStatus		:= Done;

			END_IF

		MtrPshrActSetSpdBit1:
			IF tylocalMtrPshr.Out.eStatus = Idle OR tylocalMtrPshr.Out.eStatus = Busy THEN

				tylocalMtrPshr.Out.bSpdBinBit1	:= TRUE;

				tylocalMtrPshr.Out.eStatus		:= Done;

			END_IF

		MtrPshrActRstSpdBit1:
			IF tylocalMtrPshr.Out.eStatus = Idle OR tylocalMtrPshr.Out.eStatus = Busy THEN

				tylocalMtrPshr.Out.bSpdBinBit1	:= FALSE;

				tylocalMtrPshr.Out.eStatus		:= Done;

			END_IF

		MtrPshrActSetSpdBit2:
			IF tylocalMtrPshr.Out.eStatus = Idle OR tylocalMtrPshr.Out.eStatus = Busy THEN

				tylocalMtrPshr.Out.bSpdBinBit2	:= TRUE;

				tylocalMtrPshr.Out.eStatus		:= Done;

			END_IF

		MtrPshrActRstSpdBit2:
			IF tylocalMtrPshr.Out.eStatus = Idle OR tylocalMtrPshr.Out.eStatus = Busy THEN

				tylocalMtrPshr.Out.bSpdBinBit2	:= FALSE;

				tylocalMtrPshr.Out.eStatus		:= Done;

			END_IF

		MtrPshrActSetSigOn:
			IF tylocalMtrPshr.Out.eStatus = Idle OR tylocalMtrPshr.Out.eStatus = Busy THEN

				tylocalMtrPshr.Out.bSigOn		:= TRUE;

				tylocalMtrPshr.Out.eStatus		:= Done;

			END_IF

		MtrPshrActRstSigOn:
			IF tylocalMtrPshr.Out.eStatus = Idle OR tylocalMtrPshr.Out.eStatus = Busy THEN

				tylocalMtrPshr.Out.bSigOn		:= FALSE;

				tylocalMtrPshr.Out.eStatus		:= Done;

			END_IF

		MtrPshrActSetBrake:
			IF tylocalMtrPshr.Out.eStatus = Idle OR tylocalMtrPshr.Out.eStatus = Busy THEN

				tylocalMtrPshr.Out.bBrake		:= TRUE;

				tylocalMtrPshr.Out.eStatus		:= Done;

			END_IF

		MtrPshrActRstBrake:
			IF tylocalMtrPshr.Out.eStatus = Idle OR tylocalMtrPshr.Out.eStatus = Busy THEN

				tylocalMtrPshr.Out.bBrake		:= FALSE;

				tylocalMtrPshr.Out.eStatus		:= Done;

			END_IF

		MtrPshrActSetAlmRst:
			IF tylocalMtrPshr.Out.eStatus = Idle OR tylocalMtrPshr.Out.eStatus = Busy THEN

				tylocalMtrPshr.Out.bAlmRst		:= TRUE;

				tylocalMtrPshr.Out.eStatus		:= Done;

			END_IF

		MtrPshrActRstAlmRst:
			IF tylocalMtrPshr.Out.eStatus = Idle OR tylocalMtrPshr.Out.eStatus = Busy THEN

				tylocalMtrPshr.Out.bAlmRst		:= FALSE;

				tylocalMtrPshr.Out.eStatus		:= Done;

			END_IF

		MtrPshrActSetAll:
			IF tylocalMtrPshr.Out.eStatus = Idle OR tylocalMtrPshr.Out.eStatus = Busy THEN

				tylocalMtrPshr.Out.bCW			:= TRUE;
				tylocalMtrPshr.Out.bCCW		:= TRUE;
				tylocalMtrPshr.Out.bSpdBinBit0	:= TRUE;
				tylocalMtrPshr.Out.bSpdBinBit1	:= TRUE;
				tylocalMtrPshr.Out.bSpdBinBit2	:= TRUE;
				tylocalMtrPshr.Out.bSigOn		:= TRUE;
				tylocalMtrPshr.Out.bBrake		:= TRUE;
				tylocalMtrPshr.Out.bAlmRst		:= TRUE;

				tylocalMtrPshr.Out.eStatus		:= Done;

			END_IF

		MtrPshrActRstAll:
			IF tylocalMtrPshr.Out.eStatus = Idle OR tylocalMtrPshr.Out.eStatus = Busy THEN

				tylocalMtrPshr.Out.bCW			:= FALSE;
				tylocalMtrPshr.Out.bCCW		:= FALSE;
				tylocalMtrPshr.Out.bSpdBinBit0	:= FALSE;
				tylocalMtrPshr.Out.bSpdBinBit1	:= FALSE;
				tylocalMtrPshr.Out.bSpdBinBit2	:= FALSE;
				tylocalMtrPshr.Out.bSigOn		:= FALSE;
				tylocalMtrPshr.Out.bBrake		:= FALSE;
				tylocalMtrPshr.Out.bAlmRst		:= FALSE;

				tylocalMtrPshr.Out.eStatus		:= Done;

			END_IF

	END_CASE

END_ACTION
```

#### Act_OutputConfig.st
```iecst
ACTION Act_OutputConfig:

 g_tyMtrPshr := tylocalMtrPshr.Out; // Change the Global Naming According to the Physical Hardware Module

END_ACTION
```

#### Cyclic.st
```iecst
(** 2019-03-29 **)
PROGRAM _CYCLIC

	IF bInitialDone = FALSE THEN
		IF g_tyStartUp.bNtSettingsLoadDone = TRUE THEN
			bInitialDone	:= TRUE;
			Act_Initial;
		END_IF
	ELSE
		Act_InputConfig;
		IF (tylocalMtrPshr.In.bPrep = TRUE) AND (tylocalMtrPshr.In.bEn = TRUE) AND (tylocalMtrPshr.In.bDis = FALSE) THEN
			Act_Link;
			Act_Main;
			Act_Background;
		ELSE
			IF tylocalMtrPshr.Out.eStat <> MtrPshrActIdle THEN
				tylocalMtrPshr.Out.eStatus	:= Done;
			ELSE
				tylocalMtrPshr.Out.eStatus	:= Idle;
			END_IF
		END_IF
		Act_OutputConfig;
		Act_Alarm;

	END_IF

END_PROGRAM
```

#### Init.st
```iecst
(** 2019-03-25 **)
PROGRAM _INIT

	(* Always Change If Project Change *)

	//Pass Address To Global Address For External Use
	//Action, State & Status
	p_MtrPshrStat		:= ADR(eStat);
	p_MtrPshrStatus		:= ADR(eStatus);
	p_MtrPshrStatTxt	:= ADR(sStatTxt);

	//Alarm
	p_MtrPshrAlmData	:= ADR(tyAlmData);

	//Output
	p_MtrPshrExtended	:= ADR(bExtended);
	p_MtrPshrRetracted	:= ADR(bRetracted);
	p_MtrPshrCW			:= ADR(bCW);
	p_MtrPshrCCW		:= ADR(bCCW);
	p_MtrPshrSpdBinBit0	:= ADR(bSpdBinBit0);
	p_MtrPshrSpdBinBit1	:= ADR(bSpdBinBit1);
	p_MtrPshrSpdBinBit2	:= ADR(bSpdBinBit2);
	p_MtrPshrSigOn		:= ADR(bSigOn);
	p_MtrPshrBrake		:= ADR(bBrake);
	p_MtrPshrAlmRst		:= ADR(bAlmRst);

	(* Always Change If Project Change *)

END_PROGRAM
```

### SOT.typ - Do Not Change!!!
```iecst
(*2021-04-19*)
(**)
(*Action*)

TYPE
	eSOTAction :
		(
		SOTActIdle,
		SOTActRun,
		SOTActSetSig,
		SOTActRstSig
		);
	tySOTstatus : 	STRUCT
		tyBtnInPos : BOOL;
		tyBtnError : BOOL;
		tyBtnRdy : BOOL;
		tyBtnAvail : BOOL;
	END_STRUCT;
END_TYPE

(* *)

TYPE
	tyUSSOT : 	STRUCT
		In : tyUSSOTIn1;
		Out : tyUSSOTOut1;
	END_STRUCT;
	tyUSSOTIn1 : 	STRUCT
		eAct : eConvAction;
		udiRstErr : UDINT := 0;
		bPrep : BOOL := TRUE;
		bEn : BOOL := TRUE;
		bDis : BOOL := FALSE;
		bManual : BOOL := FALSE;
		diTransferInTO : DINT := 20000;
		bDirLToR : BOOL := FALSE;
		bRdyRcv : BOOL := TRUE;
		bLeftSen : BOOL := FALSE;
		bRightSen : BOOL := FALSE;
		bComplSigOn : BOOL := FALSE;
		bUMA : BOOL := FALSE;
		bUMASize : BOOL := FALSE;
		bVirtualEn : BOOL;
		bUBAVirtual : BOOL;
		tRstDlyTm : TIME := T#500ms;
		tSigInChkTm : TIME := T#100ms;
		sProgNm : STRING[15];
		bLinkSOTReadyOnFirst : BOOL;
		bLinkProjMag1ConvPrep : BOOL;
		bLinkProjMagConvLane1Prep : BOOL;
		bLinkProjTCPAGVSigPrep : BOOL;
	END_STRUCT;
	tyUSSOTOut1 : 	STRUCT
		eStat : eConvAction;
		eStatus : eFBStatus;
		sStatTxt : STRING[200];
		tyAlmData : tyAlmDat;
		bUSRdy : BOOL := FALSE;
		bUSLargeMagRdy : BOOL := FALSE;
		bDSRdy : BOOL := FALSE;
		bTransporting : BOOL := FALSE;
		bConvStart : BOOL := FALSE;
		bConvStop : BOOL := FALSE;
		bUSB : BOOL := FALSE;
		bVirtual : BOOL;
	END_STRUCT;
END_TYPE

(**)

TYPE
	tyDSSOT : 	STRUCT
		In : tyUSSOTIn1;
		Out : tyUSSOTOut1;
	END_STRUCT;
	tyDSSOTIn1 : 	STRUCT
		eAct : eConvAction;
		udiRstErr : UDINT := 0;
		bPrep : BOOL := TRUE;
		bEn : BOOL := TRUE;
		bDis : BOOL := FALSE;
		bManual : BOOL := FALSE;
		diTransferOutTO : DINT := 20000;
		bDirLToR : BOOL := FALSE;
		bRdySend : BOOL := TRUE;
		bLeftSen : BOOL := FALSE;
		bRightSen : BOOL := FALSE;
		bComplSigOn : BOOL := FALSE;
		bMagSizeLarge : BOOL := FALSE;
		bDSB : BOOL := FALSE;
		bVirtualEn : BOOL;
		bDSBVirtual : BOOL;
		tRstDlyTm : TIME := T#500ms;
		tSigInChkTm : TIME := T#100ms;
		sProgNm : STRING[15];
		bLinkProjMag2ConvPrep : BOOL;
		bLinkProjMagConvLane2Prep : BOOL;
		bLinkProjTCPAGVSigPrep : BOOL;
	END_STRUCT;
	tyDSSOTOut1 : 	STRUCT
		eStat : eConvAction;
		eStatus : eFBStatus;
		sStatTxt : STRING[200];
		tyAlmData : tyAlmDat;
		bUSRdy : BOOL := FALSE;
		bDSMagSizeLarge : BOOL := FALSE;
		bDSRdy : BOOL := FALSE;
		bTransporting : BOOL := FALSE;
		bConvStart : BOOL := FALSE;
		bConvStop : BOOL := FALSE;
		bDBA : BOOL := FALSE;
		bVirtual : BOOL;
	END_STRUCT;
END_TYPE
```

### SOT.var - Change By Project
```iecst
(*2021-04-19*)
VAR
	g_tyUSSOT1 : tyUSSOTOut1;
	g_tyDSSOT1 : tyDSSOTOut1;
	g_tyUSSOT2 : tyUSSOTOut1;
	g_tyDSSOT2 : tyDSSOTOut1;
	g_tyUSSOT3 : tyUSSOTOut1;
	g_tyDSSOT3 : tyDSSOTOut1;
END_VAR
```

### Program Logical/SOT/USSOT1 (IEC) - 1.00.0 - NtSOT v5.00.0

#### InputRef_Link.var
```iecst
(*2021-04-20*)
(**)
VAR
	p_bLinkOpsRun : REFERENCE TO BOOL;
	p_bLinkSOTReadyOnFirst : REFERENCE TO BOOL;
END_VAR
(**)
VAR
	p_bLinkProjMag1ConvPrep : REFERENCE TO BOOL;
	p_bLinkProjMagConvLane1Prep : REFERENCE TO BOOL;
	p_bLinkProjTCPAGVSigPrep : REFERENCE TO BOOL;
END_VAR
```

#### Act_Action.st
```iecst
(**2021-04-20 **)
ACTION Act_Action:

	//Reset Error
	IF (eStatus = Error) AND bRstErr THEN
		p_eAct	:= SOTActIdle;
		eStat	:= SOTActIdle;
	END_IF

	//Set p_eAct
	IF eStatus = Idle OR eStatus = Busy OR eStatus = Done THEN
		eStat	:= p_eAct;
	END_IF

END_ACTION
```

#### Act_Alarm.st
```iecst
(** 2021-04-20 **)
ACTION Act_Alarm:

	//Error
	IF EDGEPOS(eStatus = Error) THEN

		tyAlmData.sProgNm		:= p_sProgNm;
		tyAlmData.udiCode		:= udiStatus;
		tyAlmData.eSeverity		:= AlmSeverityError;
		tyAlmData.udiRunTime	:= tyAlmData.udiRunTime + 1;
		tyAlmData.bAlm			:= TRUE;
		tyAlmData.udiModuleNum  := udiModuleNum;
		g_sUSSOTProgNm		:= p_sProgNm;
		//Get Error Message
		IF tyAlmData.udiCode < 10000 OR tyAlmData.udiCode > 10099 THEN
			tyAlmData.sAlmMsg	:= 'Unknown';
			tyAlmData.sRcyMsg	:= 'Unknown';
		ELSE
			tyAlmData.sAlmMsg	:= a_tyAlmText[tyAlmData.udiCode].sAlmText;
			tyAlmData.sRcyMsg	:= a_tyAlmText[tyAlmData.udiCode].sRcyText;
		END_IF

		sStatTxt	:= tyAlmData.sAlmMsg;

	ELSIF bRstErr AND (tyAlmData.udiCode <> 0) THEN

		tyAlmData.udiCode	:= 0;
		tyAlmData.eSeverity	:= AlmSeverityNA;
		tyAlmData.sAlmMsg	:= '';
		tyAlmData.sRcyMsg	:= '';
		tyAlmData.bAlm			:= FALSE;
		sStatTxt	:= a_sStatText[eStat];

	END_IF

END_ACTION
```

#### Act_Background.st
```iecst
(** 2021-04-20 **)
ACTION Act_Background:

	IF tylocalUSSOT.Out.bConvStart = FALSE AND tylocalUSSOT.Out.bConvStop = FALSE THEN

		IF tylocalUSSOT.In.bVirtualEn = TRUE THEN
			tylocalUSSOT.Out.bVirtual	:= TRUE;
		ELSE
			tylocalUSSOT.Out.bVirtual	:= FALSE;
		END_IF
	END_IF

	IF tylocalUSSOT.Out.bVirtual = TRUE THEN

		fbSigInChk.bNomSig	:= tylocalUSSOT.In.bUBAVirtual;
	ELSE

		fbSigInChk.bNomSig	:= tylocalUSSOT.In.bUMA;
		fbSigInChk.bMagSizeSig := tylocalUSSOT.In.bUMASize;

	END_IF

	fbSigInChk;

	tylocalUSSOT.Out.bUSRdy			:= fbSigInChk.bSigInValid;
	tylocalUSSOT.Out.bUSLargeMagRdy	:= fbSigInChk.bMagSizeLarge;

END_ACTION
```

#### Act_InitGlobal.st
```iecst
(** 2021-04-20 **)
ACTION Act_InitGlobal:

	(* Always Change If Project Change *)

	//Pass Data To Link
	p_bLinkOpsRun ACCESS p_OpsRun;
	p_bLinkSOTReadyOnFirst ACCESS p_NtParamSOTReadyOnFirst;
	p_bLinkProjMag1ConvPrep ACCESS p_NtParamProjMag1ConvPrep;
	p_bLinkProjMagConvLane1Prep ACCESS p_NtParamProjMagConvLane1Prep;
	p_bLinkProjTCPAGVSigPrep ACCESS p_NtParamProjTCPAGVSigPrep;

	//Pass Data To Internal Use
	p_udiRstErr ACCESS p_RstErrReset;
	p_bManual ACCESS p_UIMnlMod;
	p_diTransferInTO ACCESS p_McParamTranInErrDlyTm;
	p_bEn ACCESS p_McParamAGVComEn;
//	p_bVirtualEn ACCESS p_UIVSOTUSEn;
//	p_bUBAVirtual ACCESS p_UIVSOTUBA;
	p_tRstDlyTm ACCESS p_NtParamUSSOT1RstDlyTm;
	p_tSigInChkTm ACCESS p_NtParamUSSOT1SigInChkTm;
	p_sProgNm ACCESS p_NtParamUSSOT1ProgNm;
	p_bNtSettingsLoadDone ACCESS p_StartupNtSettingsLoadDone;

	(* Always Change If Project Change *)

END_ACTION
```

#### Act_Initial.st
```iecst
(** 2021-04-20 **)
ACTION Act_Initial:

	//Initial
	sStatTxt	:= a_sStatText[eStat];

	fbSOT.tRstDlyTm	:= p_tRstDlyTm;
	fbSOT(bEn := FALSE);

	fbSigInChk.tSigInChkTm	:= p_tSigInChkTm;

END_ACTION
```

#### Act_InitLocal.st
```iecst
(** 2021-04-20 **)
ACTION Act_InitLocal:

	//Input Reference Link To Local Variable
	p_eAct ACCESS ADR(eAct);
	p_udiRstErr ACCESS ADR(udiRstErr);
	p_bPrep ACCESS ADR(bPrep);
	p_bEn ACCESS ADR(bEn);
	p_bDis ACCESS ADR(bDis);
	p_bManual ACCESS ADR(bManual);
	p_diTransferInTO ACCESS ADR(diTransferInTO);
	p_bDirLToR ACCESS ADR(bDirLToR);
	p_bRdyRcv ACCESS ADR(bRdyRcv);
	p_bLeftSen ACCESS ADR(bLeftSen);
	p_bRightSen ACCESS ADR(bRightSen);
	p_bComplSigOn ACCESS ADR(bComplSigOn);
	p_bUMA ACCESS ADR(bUMA);
	p_bUMASize ACCESS ADR(bUMASize);
	p_bVirtualEn ACCESS ADR(bVirtualEn);
	p_bUBAVirtual ACCESS ADR(bUBAVirtual);
	p_tRstDlyTm ACCESS ADR(tRstDlyTm);
	p_tSigInChkTm ACCESS ADR(tSigInChkTm);
	p_sProgNm ACCESS ADR(sProgNm);
	p_bNtSettingsLoadDone ACCESS ADR(bNtSettingsLoadDone);

END_ACTION
```

#### Act_InputConfig.st
```iecst
(** 2021-04-20 **)
ACTION Act_InputConfig:

	(* Always Change If Project Change *)

	//Pass Data To Link
//	tylocalUSSOT.In.bLinkOpsRun := g_tyOpsRun;
	tylocalUSSOT.In.bLinkSOTReadyOnFirst := g_tyNtParamCurr.bSOTReadyOnFirst;
	tylocalUSSOT.In.bLinkProjMag1ConvPrep := g_tyNtParamCurr.bProjMag1ConvPrep;
	tylocalUSSOT.In.bLinkProjMagConvLane1Prep := g_tyNtParamCurr.bProjMagConvLane1Prep;
	tylocalUSSOT.In.bLinkProjTCPAGVSigPrep := g_tyNtParamCurr.bProjTCPAGVSigPrep;

	//Pass Data To Internal Use
	tylocalUSSOT.In.udiRstErr := g_tyRstErrOut.udiRstErr;
	tylocalUSSOT.In.bManual := g_tyUIOut.bOut.bManualMod;
	tylocalUSSOT.In.diTransferInTO := g_tyMcParamCurr.tTranInErrDlyTm;
	tylocalUSSOT.In.bEn := g_tyMcParamCurr.bAGVComEn;
//	tylocalUSSOT.In.bVirtualEn := g_tyUIOut.bVSOTUSEn;
//	tylocalUSSOT.In.bUBAVirtual := g_tyUIOut.bVSOTUBA;
	tylocalUSSOT.In.tRstDlyTm := g_tyNtParamCurr.bUSSOT1RstDlyTm;
	tylocalUSSOT.In.tSigInChkTm := g_tyNtParamCurr.bUSSOT1SigInChkTm;
	tylocalUSSOT.In.sProgNm := g_tyNtParamCurr.bUSSOT1ProgNm;

	(* Always Change If Project Change *)
	IF g_tyOps.bRun = TRUE THEN
		IF tylocalUSSOT.In.bLinkProjMag1ConvPrep THEN
			tylocalUSSOT.In.eAct := g_tyOpsMagConvUL1.eUSSOTAct;
		ELSE
			tylocalUSSOT.In.eAct := eAct;
		END_IF
	ELSE
		tylocalUSSOT.In.eAct := eAct;
	END_IF
END_ACTION
```

#### Act_Link.st
```iecst
(** 2021-04-20 **)
ACTION Act_Link:

		//Ready Receive
	IF tylocalUSSOT.In.bLinkProjTCPAGVSigPrep THEN
		//TCP package
		IF tylocalUSSOT.In.bLinkSOTReadyOnFirst THEN
			tylocalUSSOT.In.bRdyRcv	:= TRUE;
		ELSE
			tylocalUSSOT.In.bRdyRcv := g_tyTCP.bSvrUBA;
		END_IF
		tylocalUSSOT.In.bLeftSen := g_tyDInput.bInMagConvMidSen;
		tylocalUSSOT.In.bRightSen := g_tyDInput.bInMagConvEntSen;
		tylocalUSSOT.In.bUMA := g_tyTCP.bSvrUBA;
		tylocalUSSOT.In.bDirLToR := FALSE;
		tylocalUSSOT.In.bComplSigOn	:= tylocalUSSOT.In.bLeftSen;

	ELSE
		IF tylocalUSSOT.In.bLinkSOTReadyOnFirst THEN
			tylocalUSSOT.In.bRdyRcv	:= TRUE;
		ELSE
			tylocalUSSOT.In.bRdyRcv := g_tyDInput.bSOT1AIVAvailable;
		END_IF

		tylocalUSSOT.In.bLeftSen := g_tyDInput.bMagConvEntSen1;
		tylocalUSSOT.In.bRightSen := g_tyDInput.bMagPresentSen1;
		tylocalUSSOT.In.bUMA := g_tyDInput.bSOT1AIVAvailable;
		tylocalUSSOT.In.bUMASize := g_tyDInput.bSOT1AIVSizeLarge;
		tylocalUSSOT.In.bDirLToR := TRUE;

		tylocalUSSOT.In.bComplSigOn	:= tylocalUSSOT.In.bRightSen;
	END_IF

END_ACTION
```

#### Act_LinkAction.st
```iecst
(** 2021-04-20 **)
ACTION Act_LinkAction:

	IF p_bLinkOpsRun = TRUE THEN
		IF p_bLinkProjMag1ConvPrep THEN
			p_eAct ACCESS p_OpsMagConvUL1USSOTAct;
		ELSIF p_bLinkProjMagConvLane1Prep THEN
			p_eAct ACCESS p_OpsInMagConvUSSOTAct;
		ELSE
			p_eAct ACCESS ADR(eAct);
		END_IF
	ELSE
		p_eAct ACCESS ADR(eAct);
	END_IF

END_ACTION
```

#### Act_LinkEn.st
```iecst
(** 2021-04-20 **)
ACTION Act_LinkEn:

	//Link bPrep, bEn & bDis

END_ACTION
```

#### Act_Main.st
```iecst
(** 2021-04-20 **)
ACTION Act_Main:

	IF eStatOld <> eStat THEN
		fbSOT(bEn := FALSE);

		bTransporting	:= FALSE;
		bConvStart		:= FALSE;
		bConvStop		:= FALSE;
		bDSRdy			:= FALSE;

		IF eStatOld <> SOTActIdle
			AND eStatOld <> SOTActSetSig
			AND eStatOld <> SOTActRstSig THEN

			bUSB	:= FALSE;

		END_IF

		sStatTxt	:= a_sStatText[eStat];

		eStatOld	:= eStat;

		eStatus		:= Busy;
	END_IF

	//Main
	CASE eStat OF

		SOTActIdle:
			IF EDGENEG(p_bManual) THEN
				bUSB	:= FALSE;
			END_IF

			eStatus	:= Idle;

		SOTActRun:
			IF eStatus = Idle OR eStatus = Busy THEN

				eStatus	:= Busy;

				fbSOT.bUSRdy		:= fbSigInChk.bSigInValid;
				fbSOT.bRdyRcv		:= p_bRdyRcv;
				fbSOT.bComplSigOn	:= p_bComplSigOn;

				IF p_bDirLToR = TRUE THEN

					fbSOT.bInletSen		:= p_bLeftSen;
					fbSOT.bOutletSen	:= p_bRightSen;

				ELSE

					fbSOT.bInletSen		:= p_bRightSen;
					fbSOT.bOutletSen	:= p_bLeftSen;

				END_IF

				fbSOT.tTimeOut	:= DINT_TO_TIME(p_diTransferInTO);
				fbSOT(bEn := TRUE);

				bTransporting	:= fbSOT.bTransporting;
				bConvStart		:= fbSOT.bConvStart;
				bConvStop		:= fbSOT.bConvStop;
				bUSB			:= fbSOT.bSigToUS  AND (bVirtual = FALSE);
				bDSRdy			:= fbSOT.bSigToUS;

				IF fbSOT.udiStatus = 0 THEN
					eStatus	:= Done;
				ELSIF fbSOT.udiStatus < 65534 THEN
					eStatus		:= Error;

					IF fbSOT.udiStatus = 1200 THEN
						udiStatus	:= 10000;	//SOT Transport Time Out While Transporting
					ELSIF fbSOT.udiStatus = 1201 THEN
						udiStatus	:= 10001;	//SOT Transport Time Out After Opposite Machine Transport Finished
					ELSIF fbSOT.udiStatus = 1202 THEN
						udiStatus	:= 10002;	//SOT Transport Time Out After Current Machine Transport Finished
					ELSIF fbSOT.udiStatus = 1203 THEN
						udiStatus	:= 10003;	//SOT Transport Time Out After Both Machine Transport Finished And Waiting Outlet Sensor
					ELSE
						udiStatus	:= fbSOT.udiStatus;
					END_IF
				END_IF

			END_IF

		SOTActSetSig:
			IF eStatus = Idle OR eStatus = Busy THEN

				//Reset
				fbSOT(bEn := FALSE);

				bConvStart	:= FALSE;
				bConvStop	:= FALSE;

				bUSB	:= TRUE;
				eStatus	:= Done;

			END_IF

		SOTActRstSig:
			IF eStatus = Idle OR eStatus = Busy THEN

				//Reset
				fbSOT(bEn := FALSE);

				bConvStart	:= FALSE;
				bConvStop	:= FALSE;

				bUSB	:= FALSE;
				eStatus	:= Done;

			END_IF

	END_CASE

END_ACTION
```

#### Act_OutputConfig.st
```iecst
(** 2021-04-20 **)
ACTION Act_OutputConfig:

	g_tyUSSOT1 := tylocalUSSOT.Out; // Change the Global Naming According to the Physical Hardware Module

END_ACTION
```

#### Cyclic.st
```iecst
(** 2021-04-20 **)
PROGRAM _CYCLIC

	IF bInitialDone = FALSE THEN
		IF g_tyStartUp.bNtSettingsLoadDone = TRUE  THEN
			bInitialDone	:= TRUE;
			Act_Initial;
		END_IF

	ELSE

		Act_InputConfig;
		IF (tylocalUSSOT.In.bPrep = TRUE) AND (tylocalUSSOT.In.bEn = TRUE) AND (tylocalUSSOT.In.bDis = FALSE) THEN
			Act_Link;
			Act_Background;
			Act_Main;
		ELSE
			IF tylocalUSSOT.Out.eStat <> SOTActIdle THEN
				tylocalUSSOT.Out.eStatus	:= Done;
			ELSE
				tylocalUSSOT.Out.eStatus	:= Idle;
			END_IF
		END_IF
		Act_OutputConfig;
		Act_Alarm;

	END_IF

END_PROGRAM
```

#### Init.st
```iecst
(** 2021-04-20 **)
PROGRAM _INIT

	(* Always Change If Project Change *)

	//Pass Address To Global Address For External Use
	//Action, State & Status
	p_USSOT1Stat		:= ADR(eStat);
	p_USSOT1Status	:= ADR(eStatus);
	p_USSOT1StatTxt	:= ADR(sStatTxt);

	//Alarm
	p_USSOT1AlmData	:= ADR(tyAlmData);

	//Output
	p_USSOT1USRdy			:= ADR(bUSRdy);
	p_USSOT1USLargeMagRdy	:= ADR(bUSLargeMagRdy);
	p_USSOT1DSRdy			:= ADR(bDSRdy);
	p_USSOT1Transporting	:= ADR(bTransporting);
	p_USSOT1ConvStart		:= ADR(bConvStart);
	p_USSOT1ConvStop		:= ADR(bConvStop);
	p_USSOT1USB				:= ADR(bUSB);
	p_USSOT1Virtual			:= ADR(bVirtual);

	(* Always Change If Project Change *)

END_PROGRAM
```

### Program Logical/SOT/DSSOT1 (IEC) - 1.00.0 - NtSOT v5.00.0

#### InputRef_Link.var
```iecst
(*2021-04-20*)
(**)
VAR
	p_bLinkOpsRun : REFERENCE TO BOOL;
END_VAR
(**)
VAR
	p_bLinkProjMag1ConvPrep : REFERENCE TO BOOL;
	p_bLinkProjMagConvLane1Prep : REFERENCE TO BOOL;
	p_bLinkProjTCPAGVSigPrep : REFERENCE TO BOOL;
END_VAR
```

#### Act_Alarm.st
```iecst
(** 2021-04-20 **)
ACTION Act_Alarm:

	//Error
	IF EDGEPOS(eStatus = Error) THEN

		tyAlmData.sProgNm		:= p_sProgNm;
		tyAlmData.udiCode		:= udiStatus;
		tyAlmData.eSeverity		:= AlmSeverityError;
		tyAlmData.udiRunTime	:= tyAlmData.udiRunTime + 1;
		tyAlmData.bAlm			:= TRUE;
		tyAlmData.udiModuleNum  := udiModuleNum;
		g_sDSSOTProgNm		:= p_sProgNm;

		//Get Error Message
		IF tyAlmData.udiCode < 10000 OR tyAlmData.udiCode > 10099 THEN
			tyAlmData.sAlmMsg	:= 'Unknown';
			tyAlmData.sRcyMsg	:= 'Unknown';
		ELSE
			tyAlmData.sAlmMsg	:= a_tyAlmText[tyAlmData.udiCode].sAlmText;
			tyAlmData.sRcyMsg	:= a_tyAlmText[tyAlmData.udiCode].sRcyText;
		END_IF

		sStatTxt	:= tyAlmData.sAlmMsg;

	ELSIF bRstErr AND (tyAlmData.udiCode <> 0) THEN

		tyAlmData.udiCode	:= 0;
		tyAlmData.eSeverity	:= AlmSeverityNA;
		tyAlmData.sAlmMsg	:= '';
		tyAlmData.sRcyMsg	:= '';
		tyAlmData.bAlm			:= FALSE;
		sStatTxt	:= a_sStatText[eStat];

	END_IF

END_ACTION
```

#### Act_InitGlobal.st
```iecst
(** 2021-04-20 **)
ACTION Act_InitGlobal:

	(* Always Change If Project Change *)

	//Pass Data To Link
	p_bLinkOpsRun ACCESS p_OpsRun;
	p_bLinkProjMag1ConvPrep ACCESS p_NtParamProjMag1ConvPrep;
	p_bLinkProjMagConvLane1Prep ACCESS p_NtParamProjMagConvLane1Prep;
	p_bLinkProjTCPAGVSigPrep ACCESS p_NtParamProjTCPAGVSigPrep;

	//Pass Data To Internal Use
	p_udiRstErr ACCESS p_RstErrReset;
	p_bManual ACCESS p_UIMnlMod;
	p_diTransferOutTO ACCESS p_McParamTranInErrDlyTm;
	p_bEn ACCESS p_McParamAGVComEn;
//	p_bVirtualEn ACCESS p_UIVSOTDSEn;
//	p_bDSBVirtual ACCESS p_UIVSOTDSB;
	p_tRstDlyTm ACCESS p_NtParamDSSOT1RstDlyTm;
	p_tSigInChkTm ACCESS p_NtParamDSSOT1SigInChkTm;
	p_sProgNm ACCESS p_NtParamDSSOT1ProgNm;
	p_bNtSettingsLoadDone ACCESS p_StartupNtSettingsLoadDone;

	p_bMagSizeLarge ACCESS p_OpsMagConvUL1MagSizeL;

	(* Always Change If Project Change *)

END_ACTION
```

#### Act_Initial.st
```iecst
(** 2021-04-20 **)
ACTION Act_Initial:

	//Initial
	sStatTxt	:= a_sStatText[eStat];

	fbSOT(bEn := FALSE);

END_ACTION
```

#### Act_Link.st
```iecst
(** 2021-04-20 **)
ACTION Act_Link:

		//Ready Send
	tylocalDSSOT.In.bRdySend	:= TRUE;

	IF tylocalDSSOT.In.bLinkProjTCPAGVSigPrep THEN //TCP AGV
		tylocalDSSOT.In.bLeftSen := g_tyDInput.bOutMagConvExtSen;
		tylocalDSSOT.In.bRightSen := g_tyDInput.bOutMagConvMidSen;
		tylocalDSSOT.In.bDSB := g_tyTCPSvr.bDSB;

		//Send Complete Signal
		IF EDGENEG(tylocalDSSOT.In.bLeftSen) THEN
			tylocalDSSOT.In.bComplSigOn	:= TRUE;
		END_IF

		IF tylocalDSSOT.Out.eStat <> SOTActRun THEN
			tylocalDSSOT.In.bComplSigOn	:= FALSE;
		END_IF
	ELSE
		tylocalDSSOT.In.bLeftSen := g_tyDInput.bMagConvEntSen1;
		tylocalDSSOT.In.bRightSen := g_tyDInput.bMagPresentSen1;
		tylocalDSSOT.In.bDSB := g_tyDInput.bSOT1AIVReady;

		//Send Complete Signal
		IF EDGENEG(tylocalDSSOT.In.bLeftSen) THEN
			tylocalDSSOT.In.bComplSigOn	:= TRUE;
		END_IF

		IF tylocalDSSOT.Out.eStat <> SOTActRun THEN
			tylocalDSSOT.In.bComplSigOn	:= FALSE;
		END_IF

	END_IF

END_ACTION
```

#### Act_LinkAction.st
```iecst
(** 2021-04-20 **)
ACTION Act_LinkAction:

	IF p_bLinkOpsRun = TRUE THEN
		IF p_bLinkProjMag1ConvPrep THEN
			p_eAct ACCESS p_OpsMagConvUL1DSSOTAct;
		ELSIF p_bLinkProjMagConvLane1Prep THEN
			p_eAct ACCESS p_OpsOutMagConvDSSOTAct;
		ELSE
			p_eAct ACCESS ADR(eAct);
		END_IF
	ELSE
		p_eAct ACCESS ADR(eAct);
	END_IF

END_ACTION
```

#### Act_Main.st
```iecst
(** 2021-04-20 **)
ACTION Act_Main:

	//Main
	fbSOT.tRstDlyTm	:= tylocalDSSOT.In.tRstDlyTm;
	fbSigInChk.tSigInChkTm	:= tylocalDSSOT.In.tSigInChkTm;
	//Set tylocalDSSOT.In.eAct
	IF tylocalDSSOT.Out.eStatus = Idle OR tylocalDSSOT.Out.eStatus = Busy OR tylocalDSSOT.Out.eStatus = Done THEN
		tylocalDSSOT.Out.eStat	:= tylocalDSSOT.In.eAct;
	END_IF
	IF eStatOld <> tylocalDSSOT.Out.eStat THEN
		fbSOT(bEn := FALSE);

		tylocalDSSOT.Out.bTransporting	:= FALSE;
		tylocalDSSOT.Out.bConvStart		:= FALSE;
		tylocalDSSOT.Out.bConvStop		:= FALSE;
		tylocalDSSOT.Out.bUSRdy			:= FALSE;

		IF eStatOld <> SOTActIdle
			AND eStatOld <> SOTActSetSig
			AND eStatOld <> SOTActRstSig THEN

			tylocalDSSOT.Out.bDBA			:= FALSE;
			tylocalDSSOT.Out.bDSMagSizeLarge	:= FALSE;

		END_IF

		tylocalDSSOT.Out.sStatTxt	:= a_sStatText[tylocalDSSOT.Out.eStat];

		eStatOld	:= tylocalDSSOT.Out.eStat;

		tylocalDSSOT.Out.eStatus		:= Busy;
	END_IF

	//Main
	CASE tylocalDSSOT.Out.eStat OF

		SOTActIdle:
			IF EDGENEG(tylocalDSSOT.In.bManual) THEN
				tylocalDSSOT.Out.bDBA		:= FALSE;
				tylocalDSSOT.Out.bDSMagSizeLarge	:= FALSE;
			END_IF

			tylocalDSSOT.Out.eStatus	:= Idle;

		SOTActRun:
			IF tylocalDSSOT.Out.eStatus = Idle OR tylocalDSSOT.Out.eStatus = Busy THEN

				tylocalDSSOT.Out.eStatus	:= Busy;

				fbSOT.tylocalDSSOT.Out.bDSRdy		:= fbSigInChk.bSigInValid;
				fbSOT.bRdySend		:= tylocalDSSOT.In.bRdySend;
				fbSOT.bComplSigOn	:= tylocalDSSOT.In.bComplSigOn;

				fbSOT.tTimeOut	:= DINT_TO_TIME(tylocalDSSOT.In.diTransferOutTO);
				fbSOT(bEn := TRUE);

				tylocalDSSOT.Out.bTransporting	:= fbSOT.tylocalDSSOT.Out.bTransporting;
				tylocalDSSOT.Out.bConvStart		:= fbSOT.tylocalDSSOT.Out.bConvStart;
				tylocalDSSOT.Out.bConvStop		:= fbSOT.tylocalDSSOT.Out.bConvStop;
				tylocalDSSOT.Out.bDBA			:= fbSOT.bSigToDS AND (tylocalDSSOT.Out.bVirtual = FALSE);
				tylocalDSSOT.Out.bDSMagSizeLarge	:= tylocalDSSOT.In.bMagSizeLarge;

				tylocalDSSOT.Out.bUSRdy			:= fbSOT.bSigToDS;

				IF fbSOT.udiStatus = 0 THEN
					tylocalDSSOT.Out.eStatus	:= Done;
				ELSIF fbSOT.udiStatus < 65534 THEN
					tylocalDSSOT.Out.eStatus		:= Error;

					IF fbSOT.udiStatus = 1200 THEN
						udiStatus	:= 10000;	//SOT  Transport Time Out While Transporting
					ELSIF fbSOT.udiStatus = 1201 THEN
						udiStatus	:= 10001;	//SOT  Transport Time Out After Opposite Machine Transport Finished
					ELSIF fbSOT.udiStatus = 1202 THEN
						udiStatus	:= 10002;	//SOT  Transport Time Out After Current Machine Transport Finished
					ELSIF fbSOT.udiStatus = 1203 THEN
						udiStatus	:= 10003;	//SOT  Transport Time Out After Both Machine Transport Finished And Waiting Outlet Sensor
					ELSE
						udiStatus	:= fbSOT.udiStatus;
					END_IF
				END_IF

			END_IF

		SOTActSetSig:
			IF tylocalDSSOT.Out.eStatus = Idle OR tylocalDSSOT.Out.eStatus = Busy THEN

				//Reset
				fbSOT(bEn := FALSE);

				tylocalDSSOT.Out.bConvStart	:= FALSE;
				tylocalDSSOT.Out.bConvStop	:= FALSE;

				tylocalDSSOT.Out.bDBA	:= TRUE;
				tylocalDSSOT.Out.eStatus	:= Done;

			END_IF

		SOTActRstSig:
			IF tylocalDSSOT.Out.eStatus = Idle OR tylocalDSSOT.Out.eStatus = Busy THEN

				//Reset
				fbSOT(bEn := FALSE);

				tylocalDSSOT.Out.bConvStart	:= FALSE;
				tylocalDSSOT.Out.bConvStop	:= FALSE;

				tylocalDSSOT.Out.bDBA	:= FALSE;
				tylocalDSSOT.Out.eStatus	:= Done;

			END_IF

	END_CASE

END_ACTION
```

#### Act_OutputConfig.st
```iecst
(** 2021-04-20 **)
ACTION Act_OutputConfig:

	g_tyDSSOT1 := tylocalDSSOT.Out; // Change the Global Naming According to the Physical Hardware Module

END_ACTION
```

#### Init.st
```iecst
(** 2021-04-20 **)
PROGRAM _INIT

	(* Always Change If Project Change *)

	//Pass Address To Global Address For External Use
	//Action, State & Status
	p_DSSOT1Stat		:= ADR(eStat);
	p_DSSOT1Status		:= ADR(eStatus);
	p_DSSOT1StatTxt		:= ADR(sStatTxt);

	//Alarm
	p_DSSOT1AlmData	:= ADR(tyAlmData);

	//Output
	p_DSSOT1USRdy			:= ADR(bUSRdy);
	p_DSSOT1DSRdy			:= ADR(bDSRdy);
	p_DSSOT1Transporting	:= ADR(bTransporting);
	p_DSSOT1ConvStart		:= ADR(bConvStart);
	p_DSSOT1ConvStop		:= ADR(bConvStop);
	p_DSSOT1DBA				:= ADR(bDBA);
	p_DSSOT1Virtual			:= ADR(bVirtual);
	p_DSSOT1MagSizeLarge	:= ADR(bDSMagSizeLarge);

	(* Always Change If Project Change *)

END_PROGRAM
```

### Program Logical/SOT/USSOT2 (IEC) - 1.00.0 - NtSOT v5.00.0

#### InputRef.var
```iecst
(*2021-04-20*)
(**)
(*General*)
VAR
	p_eAct : REFERENCE TO eSOTAction;
	p_udiRstErr : REFERENCE TO UDINT;
	p_bPrep : REFERENCE TO BOOL;
	p_bEn : REFERENCE TO BOOL;
	p_bDis : REFERENCE TO BOOL;
END_VAR
(**)
(*Configuration*)
VAR
	p_bManual : REFERENCE TO BOOL;
	p_diTransferInTO : REFERENCE TO DINT;
	p_bDirLToR : REFERENCE TO BOOL;
	p_bRdyRcv : REFERENCE TO BOOL;
END_VAR
(**)
(*Input*)
VAR
	p_bLeftSen : REFERENCE TO BOOL;
	p_bRightSen : REFERENCE TO BOOL;
	p_bComplSigOn : REFERENCE TO BOOL;
	p_bUMA : REFERENCE TO BOOL;
	p_bUMASize : REFERENCE TO BOOL;
	p_bVirtualEn : REFERENCE TO BOOL;
	p_bUBAVirtual : REFERENCE TO BOOL;
	p_tRstDlyTm : REFERENCE TO TIME;
	p_tSigInChkTm : REFERENCE TO TIME;
	p_sProgNm : REFERENCE TO STRING[15];
	p_bNtSettingsLoadDone : REFERENCE TO BOOL;
END_VAR
```

#### InputRef_Link.var
```iecst
(*2021-04-20*)
(**)
VAR
	p_bLinkOpsRun : REFERENCE TO BOOL;
	p_bLinkSOTReadyOnFirst : REFERENCE TO BOOL;
END_VAR
(**)
VAR
	p_bLinkProjMag2ConvPrep : REFERENCE TO BOOL;
	p_bLinkProjMagConvLane2Prep : REFERENCE TO BOOL;
	p_bLinkProjTCPAGVSigPrep : REFERENCE TO BOOL;
END_VAR
```

#### Local.var
```iecst
(*2021-04-20*)
(**)
(*Local Action, State & Status*)
VAR
	eAct : eSOTAction := SOTActIdle;
	eStat : eSOTAction := SOTActIdle;
	eStatus : eFBStatus := Idle;
	udiStatus : UDINT := 0;
	sStatTxt : STRING[200] := '';
	a_sStatText : ARRAY[0..50] OF STRING[200] := ['Idling','Upstream SOT Running','Turning On USB Signal','Turning Off USB Signal',47('')];
END_VAR
(**)
(*Local Alarm*)
VAR
	tyAlmData : tyAlmDat;
	a_tyAlmText : ARRAY[10000..10099] OF tyAlmTxt := [(sAlmText:='SOT Transport Time Out While Transporting',sRcyText:='Timeout Expired Before Operation Completed. Reset And Resume Operation.'),(sAlmText:='SOT Transport Time Out After Opposite Machine Transport Finished',sRcyText:='Timeout Expired Before Operation Completed. Reset And Resume Operation.'),(sAlmText:='SOT Transport Time Out After Current Machine Transport Finished',sRcyText:='Timeout Expired Before Operation Completed. Reset And Resume Operation.'),(sAlmText:='SOT Transport Time Out After Both Machine Transport Finished And Waiting Outlet Sensor',sRcyText:='Timeout Expired Before Operation Completed. Reset And Resume Operation.'),96(0)];
END_VAR
(**)
(*Local Output*)
VAR
	bUSRdy : BOOL := FALSE;
	bUSLargeMagRdy : BOOL := FALSE;
	bDSRdy : BOOL := FALSE;
	bTransporting : BOOL := FALSE;
	bConvStart : BOOL := FALSE;
	bConvStop : BOOL := FALSE;
	bUSB : BOOL := FALSE;
	bVirtual : BOOL;
END_VAR
(**)
(*Local Input*)
VAR
	udiRstErr : UDINT := 0;
	bPrep : BOOL := TRUE;
	bEn : BOOL := TRUE;
	bDis : BOOL := FALSE;
	bManual : BOOL := FALSE;
	diTransferInTO : DINT := 20000;
	bDirLToR : BOOL := FALSE;
	bRdyRcv : BOOL := TRUE;
	bLeftSen : BOOL := FALSE;
	bRightSen : BOOL := FALSE;
	bComplSigOn : BOOL := FALSE;
	bUMA : BOOL := FALSE;
	bUMASize : BOOL := FALSE;
	bVirtualEn : BOOL;
	bUBAVirtual : BOOL;
	tRstDlyTm : TIME := T#500ms;
	tSigInChkTm : TIME := T#100ms;
	sProgNm : STRING[15] := 'USSOT';
	bNtSettingsLoadDone : BOOL := TRUE;
END_VAR
(**)
(*Local*)
VAR
	bRstErr : BOOL;
	udiRstErrOld : UDINT;
	bInitDone : BOOL;
	bInitialDone : BOOL;
	fbSOT : fbSOTUS;
	fbSigInChk : fbSOTSigInChk;
	eStatOld : eSOTAction := SOTActIdle;
	udiModuleNum : UDINT := 4401;
END_VAR
```

#### Act_InitGlobal.st
```iecst
(** 2021-04-20 **)
ACTION Act_InitGlobal:

	(* Always Change If Project Change *)

	//Pass Data To Link
	p_bLinkOpsRun ACCESS p_OpsRun;
	p_bLinkSOTReadyOnFirst ACCESS p_NtParamSOTReadyOnFirst;
	p_bLinkProjMag2ConvPrep ACCESS p_NtParamProjMag2ConvPrep;
	p_bLinkProjMagConvLane2Prep ACCESS p_NtParamProjMagConvLane2Prep;
	p_bLinkProjTCPAGVSigPrep ACCESS p_NtParamProjTCPAGVSigPrep;

	//Pass Data To Internal Use
	p_udiRstErr ACCESS p_RstErrReset;
	p_bManual ACCESS p_UIMnlMod;
	p_diTransferInTO ACCESS p_McParamTranInErrDlyTm;
	p_bEn ACCESS p_McParamAGVComEn;
//	p_bVirtualEn ACCESS p_UIVSOTUSEn;
//	p_bUBAVirtual ACCESS p_UIVSOTUBA;
	p_tRstDlyTm ACCESS p_NtParamUSSOT2RstDlyTm;
	p_tSigInChkTm ACCESS p_NtParamUSSOT2SigInChkTm;
	p_sProgNm ACCESS p_NtParamUSSOT2ProgNm;
	p_bNtSettingsLoadDone ACCESS p_StartupNtSettingsLoadDone;

	(* Always Change If Project Change *)

END_ACTION
```

#### Act_InputConfig.st
```iecst
(** 2022-04-20 **)
ACTION Act_InputConfig:

	(* Always Change If Project Change *)

	//Pass Data To Link
//	tylocalUSSOT.In.bLinkOpsRun := g_tyOpsRun;
	tylocalUSSOT.In.bLinkSOTReadyOnFirst := g_tyNtParamCurr.bSOTReadyOnFirst;
	tylocalUSSOT.In.bLinkProjMag2ConvPrep := g_tyNtParamCurr.bProjMag2ConvPrep;
	tylocalUSSOT.In.bLinkProjMagConvLane2Prep := g_tyNtParamCurr.bProjMagConvLane2Prep;
	tylocalUSSOT.In.bLinkProjTCPAGVSigPrep := g_tyNtParamCurr.bProjTCPAGVSigPrep;

	//Pass Data To Internal Use
	tylocalUSSOT.In.udiRstErr := g_tyRstErrOut.udiRstErr;
	tylocalUSSOT.In.bManual := g_tyUIOut.bOut.bManualMod;
	tylocalUSSOT.In.diTransferInTO := g_tyMcParamCurr.tTranInErrDlyTm;
	tylocalUSSOT.In.bEn := g_tyMcParamCurr.bAGVComEn;
//	tylocalUSSOT.In.bVirtualEn := g_tyUIOut.bVSOTUSEn;
//	tylocalUSSOT.In.bUBAVirtual := g_tyUIOut.bVSOTUBA;
	tylocalUSSOT.In.tRstDlyTm := g_tyNtParamCurr.bUSSOT2RstDlyTm;
	tylocalUSSOT.In.tSigInChkTm := g_tyNtParamCurr.bUSSOT2SigInChkTm;
	tylocalUSSOT.In.sProgNm := g_tyNtParamCurr.bUSSOT2ProgNm;

	(* Always Change If Project Change *)
	IF g_tyOps.bRun = TRUE THEN
		IF tylocalUSSOT.In.bLinkProjMag2ConvPrep THEN
			tylocalUSSOT.In.eAct := g_tyOpsMagConvUL2.eUSSOTAct;
		ELSE
			tylocalUSSOT.In.eAct := eAct;
		END_IF
	ELSE
		tylocalUSSOT.In.eAct := eAct;
	END_IF
END_ACTION
```

#### Act_Link.st
```iecst
(** 2022-04-20 **)
ACTION Act_Link:

		//Ready Receive
	IF tylocalUSSOT.In.bLinkProjTCPAGVSigPrep THEN
		//TCP package
		IF tylocalUSSOT.In.bLinkSOTReadyOnFirst THEN
			tylocalUSSOT.In.bRdyRcv	:= TRUE;
		ELSE
			tylocalUSSOT.In.bRdyRcv := g_tyTCP.bSvrUBA;
		END_IF
		tylocalUSSOT.In.bLeftSen := g_tyDInput.bInMagConvMidSen;
		tylocalUSSOT.In.bRightSen := g_tyDInput.bInMagConvEntSen;
		tylocalUSSOT.In.bUMA := g_tyTCP.bSvrUBA;
		tylocalUSSOT.In.bDirLToR := FALSE;
		tylocalUSSOT.In.bComplSigOn	:= tylocalUSSOT.In.bLeftSen;

	ELSE
		IF tylocalUSSOT.In.bLinkSOTReadyOnFirst THEN
			tylocalUSSOT.In.bRdyRcv	:= TRUE;
		ELSE
			tylocalUSSOT.In.bRdyRcv := g_tyDInput.bSOT2AIVAvailable;
		END_IF

		tylocalUSSOT.In.bLeftSen := g_tyDInput.bMagConvEntSen2;
		tylocalUSSOT.In.bRightSen := g_tyDInput.bMagPresentSen2;
		tylocalUSSOT.In.bUMA := g_tyDInput.bSOT2AIVAvailable;
		tylocalUSSOT.In.bUMASize := g_tyDInput.bSOT2AIVSizeLarge;
		tylocalUSSOT.In.bDirLToR := TRUE;

		tylocalUSSOT.In.bComplSigOn	:= tylocalUSSOT.In.bRightSen;
	END_IF

END_ACTION
```

#### Act_LinkAction.st
```iecst
(** 2021-04-20 **)
ACTION Act_LinkAction:

	IF p_bLinkOpsRun = TRUE THEN
		IF p_bLinkProjMag2ConvPrep THEN
			p_eAct ACCESS p_OpsMagConvUL2USSOTAct;
		ELSIF p_bLinkProjMagConvLane2Prep THEN
			p_eAct ACCESS p_OpsInMagConv2USSOTAct;
		ELSE
			p_eAct ACCESS ADR(eAct);
		END_IF
	ELSE
		p_eAct ACCESS ADR(eAct);
	END_IF

END_ACTION
```

#### Act_OutputConfig.st
```iecst
(** 2021-04-20 **)
ACTION Act_OutputConfig:

	g_tyUSSOT2 := tylocalUSSOT.Out; // Change the Global Naming According to the Physical Hardware Module

END_ACTION
```

#### Cyclic.st
```iecst
(** 2021-04-20 **)
PROGRAM _CYCLIC

	IF bInitDone = FALSE THEN
		bInitDone	:= TRUE;

		Act_InitLocal;
		Act_InitGlobal;

	ELSIF bInitialDone = FALSE THEN
		IF p_bNtSettingsLoadDone = TRUE THEN
			bInitialDone	:= TRUE;

			Act_Initial;
		END_IF

	ELSE

		Act_RstErr;
		Act_LinkAction;
		Act_Action;
		Act_LinkEn;

		IF (p_bPrep = TRUE) AND (p_bEn = TRUE) AND (p_bDis = FALSE) THEN
			Act_Link;
			Act_Background;
			Act_Main;
		ELSE
			IF eStat <> SOTActIdle THEN
				eStatus	:= Done;
			ELSE
				eStatus	:= Idle;
			END_IF
		END_IF

		Act_Alarm;

	END_IF

END_PROGRAM
```

#### Init.st
```iecst
(** 2021-04-20 **)
PROGRAM _INIT

	(* Always Change If Project Change *)

	//Pass Address To Global Address For External Use
	//Action, State & Status
	p_USSOT2Stat		:= ADR(eStat);
	p_USSOT2Status	:= ADR(eStatus);
	p_USSOT2StatTxt	:= ADR(sStatTxt);

	//Alarm
	p_USSOT2AlmData	:= ADR(tyAlmData);

	//Output
	p_USSOT2USRdy			:= ADR(bUSRdy);
	p_USSOT2USLargeMagRdy	:= ADR(bUSLargeMagRdy);
	p_USSOT2DSRdy			:= ADR(bDSRdy);
	p_USSOT2Transporting	:= ADR(bTransporting);
	p_USSOT2ConvStart		:= ADR(bConvStart);
	p_USSOT2ConvStop		:= ADR(bConvStop);
	p_USSOT2USB				:= ADR(bUSB);
	p_USSOT2Virtual			:= ADR(bVirtual);

	(* Always Change If Project Change *)

END_PROGRAM
```

### Program Logical/SOT/DSSOT2 (IEC) - 1.00.0 - NtSOT v5.00.0

#### InputRef_Link.var
```iecst
(*2021-04-20*)
(**)
VAR
	p_bLinkOpsRun : REFERENCE TO BOOL;
END_VAR
(**)
VAR
	p_bLinkProjMag2ConvPrep : REFERENCE TO BOOL;
	p_bLinkProjMagConvLane2Prep : REFERENCE TO BOOL;
	p_bLinkProjTCPAGVSigPrep : REFERENCE TO BOOL;
END_VAR
```

#### Act_Alarm.st
```iecst
(** 2021-04-20 **)
ACTION Act_Alarm:

	//Error
	IF EDGEPOS(eStatus = Error) THEN

		tyAlmData.sProgNm		:= p_sProgNm;
		tyAlmData.udiCode		:= udiStatus;
		tyAlmData.eSeverity		:= AlmSeverityError;
		tyAlmData.udiRunTime	:= tyAlmData.udiRunTime + 1;
		tyAlmData.bAlm			:= TRUE;
		tyAlmData.udiModuleNum  := udiModuleNum;
		g_sDSSOTProgNm		:= p_sProgNm;

		//Get Error Message
		IF tyAlmData.udiCode < 10000 OR tyAlmData.udiCode > 10099 THEN
			tyAlmData.sAlmMsg	:= 'Unknown';
			tyAlmData.sRcyMsg	:= 'Unknown';
		ELSE
			tyAlmData.sAlmMsg	:= a_tyAlmText[tyAlmData.udiCode].sAlmText;
			tyAlmData.sRcyMsg	:= a_tyAlmText[tyAlmData.udiCode].sRcyText;
		END_IF

		sStatTxt	:= tyAlmData.sAlmMsg;

	ELSIF bRstErr AND (tyAlmData.udiCode <> 0) THEN

		tyAlmData.udiCode	:= 0;
		tyAlmData.eSeverity	:= AlmSeverityNA;
		tyAlmData.sAlmMsg	:= '';
		tyAlmData.sRcyMsg	:= '';
		tyAlmData.bAlm			:= FALSE;
		sStatTxt	:= a_sStatText[eStat];

	END_IF

END_ACTION
```

#### Act_Background.st
```iecst
(** 2021-04-20 **)
ACTION Act_Background:

	//background
	IF tylocalDSSOT.Out.bConvStart = FALSE AND tylocalDSSOT.Out.bConvStop = FALSE THEN
		IF tylocalDSSOT.In.bVirtualEn = TRUE THEN
			tylocalDSSOT.Out.bVirtual	:= TRUE;
		ELSE
			tylocalDSSOT.Out.bVirtual	:= FALSE;
		END_IF
	END_IF

	IF tylocalDSSOT.Out.bVirtual = TRUE THEN

		fbSigInChk.bNomSig			:= tylocalDSSOT.In.bDSBVirtual;

	ELSE

		fbSigInChk.bNomSig			:= tylocalDSSOT.In.bDSB;

	END_IF

	fbSigInChk;

	tylocalDSSOT.Out.bDSRdy	:= fbSigInChk.bSigInValid;

END_ACTION
```

#### Act_InitGlobal.st
```iecst
(** 2021-04-20 **)
ACTION Act_InitGlobal:

	(* Always Change If Project Change *)

	//Pass Data To Link
	p_bLinkOpsRun ACCESS p_OpsRun;
	p_bLinkProjMag2ConvPrep ACCESS p_NtParamProjMag2ConvPrep;
	p_bLinkProjMagConvLane2Prep ACCESS p_NtParamProjMagConvLane2Prep;
	p_bLinkProjTCPAGVSigPrep ACCESS p_NtParamProjTCPAGVSigPrep;

	//Pass Data To Internal Use
	p_udiRstErr ACCESS p_RstErrReset;
	p_bManual ACCESS p_UIMnlMod;
	p_diTransferOutTO ACCESS p_McParamTranInErrDlyTm;
	p_bEn ACCESS p_McParamAGVComEn;
//	p_bVirtualEn ACCESS p_UIVSOTDSEn;
//	p_bDSBVirtual ACCESS p_UIVSOTDSB;
	p_tRstDlyTm ACCESS p_NtParamDSSOT2RstDlyTm;
	p_tSigInChkTm ACCESS p_NtParamDSSOT2SigInChkTm;
	p_sProgNm ACCESS p_NtParamDSSOT2ProgNm;
	p_bNtSettingsLoadDone ACCESS p_StartupNtSettingsLoadDone;

	p_bMagSizeLarge ACCESS p_OpsMagConvUL2MagSizeL;

	(* Always Change If Project Change *)

END_ACTION
```

#### Act_InitLocal.st
```iecst
(** 2021-04-20 **)
ACTION Act_InitLocal:

	//Input Reference Link To Local Variable
	p_eAct ACCESS ADR(eAct);
	p_udiRstErr ACCESS ADR(udiRstErr);
	p_bPrep ACCESS ADR(bPrep);
	p_bEn ACCESS ADR(bEn);
	p_bDis ACCESS ADR(bDis);
	p_bManual ACCESS ADR(bManual);
	p_diTransferOutTO ACCESS ADR(diTransferOutTO);
	p_bDirLToR ACCESS ADR(bDirLToR);
	p_bRdySend ACCESS ADR(bRdySend);
	p_bLeftSen ACCESS ADR(bLeftSen);
	p_bRightSen ACCESS ADR(bRightSen);
	p_bComplSigOn ACCESS ADR(bComplSigOn);
	p_bDSB ACCESS ADR(bDSB);
	p_bVirtualEn ACCESS ADR(bVirtualEn);
	p_bDSBVirtual ACCESS ADR(bDSBVirtual);
	p_tRstDlyTm ACCESS ADR(tRstDlyTm);
	p_tSigInChkTm ACCESS ADR(tSigInChkTm);
	p_sProgNm ACCESS ADR(sProgNm);
	p_bNtSettingsLoadDone ACCESS ADR(bNtSettingsLoadDone);

	p_bMagSizeLarge ACCESS ADR(bMagSizeLarge);

END_ACTION
```

#### Act_InputConfig.st
```iecst
(** 2021-04-20 **)
ACTION Act_InputConfig:

	(* Always Change If Project Change *)

	//Pass Data To Link

	tylocalDSSOT.In.bLinkProjMag1ConvPrep := g_tyNtParamCurr.bProjMag1ConvPrep;
	tylocalDSSOT.In.bLinkProjMagConvLane1Prep := g_tyNtParamCurr.bProjMagConvLane1Prep;
	tylocalDSSOT.In.bLinkProjTCPAGVSigPrep := g_tyNtParamCurr.bProjTCPAGVSigPrep;

	//Pass Data To Internal Use
	tylocalDSSOT.In.udiRstErr := g_tyRstErrOut.udiRstErr;
	tylocalDSSOT.In.bManual := g_tyUIOut.bManuallMod;
	tylocalDSSOT.In.diTransferOutTO := g_tyMcParamCurr.tTranInErrDlyTm;
	tylocalDSSOT.In.bEn := g_tyMcParamCurr.bAGVComEn;
//	tylocalDSSOT.In.bVirtualEn := g_tyUIVSOTDSEn;
//	tylocalDSSOT.In.bDSBVirtual := g_tyUIVSOTDSB;
	tylocalDSSOT.In.tRstDlyTm := g_tyNtParamCurr.tDSSOT1RstDlyTm;
	tylocalDSSOT.In.tSigInChkTm := g_tyNtParamCurr.tDSSOT1SigInChkTm;
	tylocalDSSOT.In.sProgNm := g_tyNtParamCurr.sDSSOT1ProgNm;

	tylocalDSSOT.In.bMagSizeLarge := g_tyOpsMagConvUL1.bMagSizeL;

	(* Always Change If Project Change *)
	IF tylocalDSSOT.In.bLinkOpsRun = TRUE THEN
		IF tylocalDSSOT.In.bLinkProjMag1ConvPrep THEN
			tylocalDSSOT.In.eAct := g_tyOpsMagConvUL1DSSOTAct;
		ELSIF tylocalDSSOT.In.bLinkProjMagConvLane1Prep THEN
			tylocalDSSOT.In.eAct := g_tyOpsOutMagConvDSSOTAct;
		ELSE
			tylocalDSSOT.In.eAct := eAct ;
		END_IF
	ELSE
		tylocalDSSOT.In.eAct := eAct ;
	END_IF
END_ACTION
```

#### Act_Link.st
```iecst
(** 2022-04-20 **)
ACTION Act_Link:

		//Ready Send
	tylocalDSSOT.In.bRdySend	:= TRUE;

	IF tylocalDSSOT.In.bLinkProjTCPAGVSigPrep THEN //TCP AGV
		tylocalDSSOT.In.bLeftSen := g_tyDInput.bOutMagConvExtSen;
		tylocalDSSOT.In.bRightSen := g_tyDInput.bOutMagConvMidSen;
		tylocalDSSOT.In.bDSB := g_tyTCPSvr.bDSB;

		//Send Complete Signal
		IF EDGENEG(tylocalDSSOT.In.bLeftSen) THEN
			tylocalDSSOT.In.bComplSigOn	:= TRUE;
		END_IF

		IF tylocalDSSOT.Out.eStat <> SOTActRun THEN
			tylocalDSSOT.In.bComplSigOn	:= FALSE;
		END_IF
	ELSE
		tylocalDSSOT.In.bLeftSen := g_tyDInput.bMagConvEntSen2;
		tylocalDSSOT.In.bRightSen := g_tyDInput.bMagPresentSen2;
		tylocalDSSOT.In.bDSB := g_tyDInput.bSOT2AIVReady;

		//Send Complete Signal
		IF EDGENEG(tylocalDSSOT.In.bLeftSen) THEN
			tylocalDSSOT.In.bComplSigOn	:= TRUE;
		END_IF

		IF tylocalDSSOT.Out.eStat <> SOTActRun THEN
			tylocalDSSOT.In.bComplSigOn	:= FALSE;
		END_IF

	END_IF

END_ACTION
```

#### Act_LinkAction.st
```iecst
(** 2021-04-20 **)
ACTION Act_LinkAction:

	IF p_bLinkOpsRun = TRUE THEN
		IF 	p_bLinkProjMag2ConvPrep THEN
			p_eAct ACCESS p_OpsMagConvUL2DSSOTAct;
		ELSIF p_bLinkProjMagConvLane2Prep THEN
			p_eAct ACCESS p_OpsOutMagConv2DSSOTAct;
		ELSE
			p_eAct ACCESS ADR(eAct);
		END_IF
	ELSE
		p_eAct ACCESS ADR(eAct);
	END_IF

END_ACTION
```

#### Act_OutputConfig.st
```iecst
(** 2021-04-20 **)
ACTION Act_OutputConfig:

	g_tyDSSOT2 := tylocalDSSOT.Out; // Change the Global Naming According to the Physical Hardware Module

END_ACTION
```

#### Init.st
```iecst
(** 2021-04-20 **)
PROGRAM _INIT

	(* Always Change If Project Change *)

	//Pass Address To Global Address For External Use
	//Action, State & Status
	p_DSSOT2Stat		:= ADR(eStat);
	p_DSSOT2Status		:= ADR(eStatus);
	p_DSSOT2StatTxt		:= ADR(sStatTxt);

	//Alarm
	p_DSSOT2AlmData	:= ADR(tyAlmData);

	//Output
	p_DSSOT2USRdy			:= ADR(bUSRdy);
	p_DSSOT2DSRdy			:= ADR(bDSRdy);
	p_DSSOT2Transporting	:= ADR(bTransporting);
	p_DSSOT2ConvStart		:= ADR(bConvStart);
	p_DSSOT2ConvStop		:= ADR(bConvStop);
	p_DSSOT2DBA				:= ADR(bDBA);
	p_DSSOT2Virtual			:= ADR(bVirtual);
	p_DSSOT2MagSizeLarge	:= ADR(bDSMagSizeLarge);

	(* Always Change If Project Change *)

END_PROGRAM
```

### Program Logical/SOT/USSOT3 (IEC) - 1.00.0 - NtSOT v5.00.0

#### InputRef_Link.var
```iecst
(*2021-04-20*)
(**)
VAR
	p_bLinkOpsRun : REFERENCE TO BOOL;
	p_bLinkSOTReadyOnFirst : REFERENCE TO BOOL;
END_VAR
(**)
```

#### Local.var
```iecst
(*2021-04-20*)
VAR
	tylocalUSSOT : tyUSSOT;
END_VAR
(**)
(*Local Action, State & Status*)
VAR
	eAct : eSOTAction;
	udiStatus : UDINT := 0;
	a_sStatText : ARRAY[0..50] OF STRING[200] := ['Idling','Upstream SOT Running','Turning On USB Signal','Turning Off USB Signal',47('')];
END_VAR
(**)
(**)
(**)
(*Local*)
VAR
	bRstErr : BOOL;
	udiRstErrOld : UDINT;
	bInitDone : BOOL;
	bInitialDone : BOOL;
	fbSOT : fbSOTUS;
	fbSigInChk : fbSOTSigInChk;
	eStatOld : eSOTAction := SOTActIdle;
	udiModuleNum : UDINT := 4401;
END_VAR
```

#### Act_Alarm.st
```iecst
(** 2021-04-20 **)
ACTION Act_Alarm:
		//Reset Error
	IF (tylocalUSSOT.Out.eStatus = Error) AND bRstErr THEN
		tylocalUSSOT.In.eAct	:= MagConv2ClpActIdle;
		tylocalUSSOT.Out.eStat	:= MagConv2ClpActIdle;
	END_IF

	IF tylocalUSSOT.In.udiRstErr <> udiRstErrOld THEN
		bRstErr			:= TRUE;
		udiRstErrOld	:= tylocalUSSOT.In.udiRstErr;
	ELSE
		bRstErr			:= FALSE;
	END_IF
	//Error
	IF EDGEPOS(tylocalUSSOT.Out.eStatus = Error) THEN

		tylocalUSSOT.Out.tyAlmData.udiCode		:= udiStatus;
		tylocalUSSOT.Out.tyAlmData.eSeverity		:= AlmSeverityError;
		tylocalUSSOT.Out.tyAlmData.udiRunTime	:= tylocalUSSOT.Out.tyAlmData.udiRunTime + 1;
		tylocalUSSOT.Out.tyAlmData.bAlm			:= TRUE;
		tylocalUSSOT.Out.tyAlmData.udiModuleNum  := udiModuleNum;
		g_sUSSOTProgNm		    := tylocalUSSOT.In.sProgNm;

		tylocalUSSOT.Out.sStatTxt	:= tylocalUSSOT.Out.tyAlmData.sAlmMsg;

	ELSIF bRstErr AND (tyAlmData.udiCode <> 0) THEN

		tylocalUSSOT.Out.tyAlmData.udiCode	:= 0;
		tylocalUSSOT.Out.tyAlmData.eSeverity	:= AlmSeverityNA;
		tylocalUSSOT.Out.tyAlmData.bAlm			:= FALSE;
		tylocalUSSOT.Out.sStatTxt	:= a_sStatText[tylocalUSSOT.Out.eStat];

	END_IF

END_ACTION
```

#### Act_Background.st
```iecst
(** 2021-04-20 **)
ACTION Act_Background:

	IF tylocalUSSOT.Out.bConvStart = FALSE AND tylocalUSSOT.Out.bConvStop = FALSE THEN

		IF tylocalUSSOT.In.tylocalUSSOT.Out.bVirtualEn = TRUE THEN
			tylocalUSSOT.Out.bVirtual	:= TRUE;
		ELSE
			tylocalUSSOT.Out.bVirtual	:= FALSE;
		END_IF
	END_IF

	IF tylocalUSSOT.Out.bVirtual = TRUE THEN

		fbSigInChk.bNomSig	:= tylocalUSSOT.In.bUBAVirtual;
	ELSE

		fbSigInChk.bNomSig	:= tylocalUSSOT.In.bUMA;
		fbSigInChk.bMagSizeSig := tylocalUSSOT.In.bUMASize;

	END_IF

	fbSigInChk;

	tylocalUSSOT.Out.bUSRdy			:= fbSigInChk.bSigInValid;
	tylocalUSSOT.Out.bUSLargeMagRdy	:= fbSigInChk.bMagSizeLarge;

END_ACTION
```

#### Act_InitGlobal.st
```iecst
(** 2021-04-20 **)
ACTION Act_InitGlobal:

	(* Always Change If Project Change *)

	//Pass Data To Link
	p_bLinkOpsRun ACCESS p_OpsRun;
	p_bLinkSOTReadyOnFirst ACCESS p_NtParamSOTReadyOnFirst;

	//Pass Data To Internal Use
	p_udiRstErr ACCESS p_RstErrReset;
	p_bManual ACCESS p_UIMnlMod;
	p_diTransferInTO ACCESS p_McParamTranInErrDlyTm;
	p_bEn ACCESS p_McParamAGVComEn;
//	p_bVirtualEn ACCESS p_UIVSOTUSEn;
//	p_bUBAVirtual ACCESS p_UIVSOTUBA;
	p_tRstDlyTm ACCESS p_NtParamUSSOT3RstDlyTm;
	p_tSigInChkTm ACCESS p_NtParamUSSOT3SigInChkTm;
	p_sProgNm ACCESS p_NtParamUSSOT3ProgNm;
	p_bNtSettingsLoadDone ACCESS p_StartupNtSettingsLoadDone;

	(* Always Change If Project Change *)

END_ACTION
```

#### Act_InputConfig.st
```iecst
(** 2023-04-20 **)
ACTION Act_InputConfig:

	(* Always Change If Project Change *)

	//Pass Data To Link
//	tylocalUSSOT.In.bLinkOpsRun := g_tyOpsRun;
	tylocalUSSOT.In.bLinkSOTReadyOnFirst := g_tyNtParamCurr.bSOTReadyOnFirst;
	tylocalUSSOT.In.bLinkProjMag3ConvPrep := g_tyNtParamCurr.bProjMag3ConvPrep;
	tylocalUSSOT.In.bLinkProjMagConvLane3Prep := g_tyNtParamCurr.bProjMagConvLane3Prep;
	tylocalUSSOT.In.bLinkProjTCPAGVSigPrep := g_tyNtParamCurr.bProjTCPAGVSigPrep;

	//Pass Data To Internal Use
	tylocalUSSOT.In.udiRstErr := g_tyRstErrOut.udiRstErr;
	tylocalUSSOT.In.bManual := g_tyUIOut.bOut.bManualMod;
	tylocalUSSOT.In.diTransferInTO := g_tyMcParamCurr.tTranInErrDlyTm;
	tylocalUSSOT.In.bEn := g_tyMcParamCurr.bAGVComEn;
//	tylocalUSSOT.In.bVirtualEn := g_tyUIOut.bVSOTUSEn;
//	tylocalUSSOT.In.bUBAVirtual := g_tyUIOut.bVSOTUBA;
	tylocalUSSOT.In.tRstDlyTm := g_tyNtParamCurr.bUSSOT3RstDlyTm;
	tylocalUSSOT.In.tSigInChkTm := g_tyNtParamCurr.bUSSOT3SigInChkTm;
	tylocalUSSOT.In.sProgNm := g_tyNtParamCurr.bUSSOT3ProgNm;

	(* Always Change If Project Change *)
	IF g_tyOps.bRun = TRUE THEN
		IF tylocalUSSOT.In.bLinkProjMag3ConvPrep THEN
			tylocalUSSOT.In.eAct := g_tyOpsMagConvUL3.eUSSOTAct;
		ELSE
			tylocalUSSOT.In.eAct := eAct;
		END_IF
	ELSE
		tylocalUSSOT.In.eAct := eAct;
	END_IF
END_ACTION
```

#### Act_Link.st
```iecst
(** 2023-04-20 **)
ACTION Act_Link:
		//Ready Receive
	IF tylocalUSSOT.In.bLinkProjTCPAGVSigPrep THEN
		//TCP package
		IF tylocalUSSOT.In.bLinkSOTReadyOnFirst THEN
			tylocalUSSOT.In.bRdyRcv	:= TRUE;
		ELSE
			tylocalUSSOT.In.bRdyRcv := g_tyTCP.bSvrUBA;
		END_IF
		tylocalUSSOT.In.bLeftSen := g_tyDInput.bInMagConvMidSen;
		tylocalUSSOT.In.bRightSen := g_tyDInput.bInMagConvEntSen;
		tylocalUSSOT.In.bUMA := g_tyTCP.bSvrUBA;
		tylocalUSSOT.In.bDirLToR := FALSE;
		tylocalUSSOT.In.bComplSigOn	:= tylocalUSSOT.In.bLeftSen;

	ELSE
		IF tylocalUSSOT.In.bLinkSOTReadyOnFirst THEN
			tylocalUSSOT.In.bRdyRcv	:= TRUE;
		ELSE
			tylocalUSSOT.In.bRdyRcv := g_tyDInput.bSOT3AIVAvailable;
		END_IF

		tylocalUSSOT.In.bLeftSen := g_tyDInput.bMagConvEntSen3;
		tylocalUSSOT.In.bRightSen := g_tyDInput.bMagPresentSen3;
		tylocalUSSOT.In.bUMA := g_tyDInput.bSOT3AIVAvailable;
		tylocalUSSOT.In.bUMASize := g_tyDInput.bSOT3AIVSizeLarge;
		tylocalUSSOT.In.bDirLToR := TRUE;

		tylocalUSSOT.In.bComplSigOn	:= tylocalUSSOT.In.bRightSen;
	END_IF
END_ACTION
```

#### Act_LinkAction.st
```iecst
(** 2021-04-20 **)
ACTION Act_LinkAction:

	IF p_bLinkOpsRun = TRUE THEN
		p_eAct ACCESS p_OpsMagConvUL3USSOTAct;
	ELSE
		p_eAct ACCESS ADR(eAct);
	END_IF

END_ACTION
```

#### Act_Main.st
```iecst
(** 2021-04-20 **)
ACTION Act_Main:

	//Set tylocalUSSOT.In.eAct
	IF tylocalUSSOT.Out.eStatus = Idle OR tylocalUSSOT.Out.eStatus = Busy OR tylocalUSSOT.Out.eStatus = Done THEN
		tylocalUSSOT.Out.eStat	:= tylocalUSSOT.In.eAct;
	END_IF
	IF eStatOld <> tylocalUSSOT.Out.eStat THEN
		fbSOT(bEn := FALSE);

		tylocalUSSOT.Out.bTransporting	:= FALSE;
		tylocalUSSOT.Out.bConvStart		:= FALSE;
		tylocalUSSOT.Out.bConvStop		:= FALSE;
		tylocalUSSOT.Out.bDSRdy			:= FALSE;

		IF eStatOld <> SOTActIdle
			AND eStatOld <> SOTActSetSig
			AND eStatOld <> SOTActRstSig THEN

			tylocalUSSOT.Out.bUSB	:= FALSE;

		END_IF

		tylocalUSSOT.Out.sStatTxt	:= a_sStatText[tylocalUSSOT.Out.eStat];

		eStatOld	:= tylocalUSSOT.Out.eStat;

		tylocalUSSOT.Out.eStatus		:= Busy;
	END_IF

	//Main
	CASE tylocalUSSOT.Out.eStat OF

		SOTActIdle:
			IF EDGENEG(tylocalUSSOT.In.bManual) THEN
				tylocalUSSOT.Out.bUSB	:= FALSE;
			END_IF

			tylocalUSSOT.Out.eStatus	:= Idle;

		SOTActRun:
			IF tylocalUSSOT.Out.eStatus = Idle OR tylocalUSSOT.Out.eStatus = Busy THEN

				tylocalUSSOT.Out.eStatus	:= Busy;

				fbSOT.tylocalUSSOT.Out.bUSRdy		:= fbSigInChk.bSigInValid;
				fbSOT.bRdyRcv		:= tylocalUSSOT.In.bRdyRcv;
				fbSOT.bComplSigOn	:= tylocalUSSOT.In.bComplSigOn;

				IF tylocalUSSOT.In.bDirLToR = TRUE THEN

					fbSOT.bInletSen		:= tylocalUSSOT.In.bLeftSen;
					fbSOT.bOutletSen	:= tylocalUSSOT.In.bRightSen;

				ELSE

					fbSOT.bInletSen		:= tylocalUSSOT.In.bRightSen;
					fbSOT.bOutletSen	:= tylocalUSSOT.In.bLeftSen;

				END_IF

				fbSOT.tTimeOut	:= DINT_TO_TIME(tylocalUSSOT.In.diTransferInTO);
				fbSOT(bEn := TRUE);

				tylocalUSSOT.Out.bTransporting	:= fbSOT.tylocalUSSOT.Out.bTransporting;
				tylocalUSSOT.Out.bConvStart		:= fbSOT.tylocalUSSOT.Out.bConvStart;
				tylocalUSSOT.Out.bConvStop		:= fbSOT.tylocalUSSOT.Out.bConvStop;
				tylocalUSSOT.Out.bUSB			:= fbSOT.bSigToUS  AND (tylocalUSSOT.Out.bVirtual = FALSE);
				tylocalUSSOT.Out.bDSRdy			:= fbSOT.bSigToUS;

				IF fbSOT.udiStatus = 0 THEN
					tylocalUSSOT.Out.eStatus	:= Done;
				ELSIF fbSOT.udiStatus < 65534 THEN
					tylocalUSSOT.Out.eStatus		:= Error;

					IF fbSOT.udiStatus = 1200 THEN
						udiStatus	:= 10000;	//SOT Transport Time Out While Transporting
					ELSIF fbSOT.udiStatus = 1201 THEN
						udiStatus	:= 10001;	//SOT Transport Time Out After Opposite Machine Transport Finished
					ELSIF fbSOT.udiStatus = 1202 THEN
						udiStatus	:= 10002;	//SOT Transport Time Out After Current Machine Transport Finished
					ELSIF fbSOT.udiStatus = 1203 THEN
						udiStatus	:= 10003;	//SOT Transport Time Out After Both Machine Transport Finished And Waiting Outlet Sensor
					ELSE
						udiStatus	:= fbSOT.udiStatus;
					END_IF
				END_IF

			END_IF

		SOTActSetSig:
			IF tylocalUSSOT.Out.eStatus = Idle OR tylocalUSSOT.Out.eStatus = Busy THEN

				//Reset
				fbSOT(bEn := FALSE);

				tylocalUSSOT.Out.bConvStart	:= FALSE;
				tylocalUSSOT.Out.bConvStop	:= FALSE;

				tylocalUSSOT.Out.bUSB	:= TRUE;
				tylocalUSSOT.Out.eStatus	:= Done;

			END_IF

		SOTActRstSig:
			IF tylocalUSSOT.Out.eStatus = Idle OR tylocalUSSOT.Out.eStatus = Busy THEN

				//Reset
				fbSOT(bEn := FALSE);

				tylocalUSSOT.Out.bConvStart	:= FALSE;
				tylocalUSSOT.Out.bConvStop	:= FALSE;

				tylocalUSSOT.Out.bUSB	:= FALSE;
				tylocalUSSOT.Out.eStatus	:= Done;

			END_IF

	END_CASE

END_ACTION
```

#### Act_OutputConfig.st
```iecst
(** 2021-04-20 **)
ACTION Act_OutputConfig:

	g_tyUSSOT3 := tylocalUSSOT.Out; // Change the Global Naming According to the Physical Hardware Module

END_ACTION
```

#### Init.st
```iecst
(** 2021-04-20 **)
PROGRAM _INIT

	(* Always Change If Project Change *)

	//Pass Address To Global Address For External Use
	//Action, State & Status
	p_USSOT3Stat		:= ADR(eStat);
	p_USSOT3Status	:= ADR(eStatus);
	p_USSOT3StatTxt	:= ADR(sStatTxt);

	//Alarm
	p_USSOT3AlmData	:= ADR(tyAlmData);

	//Output
	p_USSOT3USRdy			:= ADR(bUSRdy);
	p_USSOT3USLargeMagRdy	:= ADR(bUSLargeMagRdy);
	p_USSOT3DSRdy			:= ADR(bDSRdy);
	p_USSOT3Transporting	:= ADR(bTransporting);
	p_USSOT3ConvStart		:= ADR(bConvStart);
	p_USSOT3ConvStop		:= ADR(bConvStop);
	p_USSOT3USB				:= ADR(bUSB);
	p_USSOT3Virtual			:= ADR(bVirtual);

	(* Always Change If Project Change *)

END_PROGRAM
```

### Program Logical/SOT/DSSOT3 (IEC, version 1.00.0) - 1.00.0 - NtSOT v5.00.0

#### Act_OutputConfig.st - Change By Project
```iecst
(** 2021-04-20 **)
ACTION Act_OutputConfig:

	g_tyDSSOT3 := tylocalDSSOT.Out; // Change the Global Naming According to the Physical Hardware Module

END_ACTION
```

#### Cyclic.st - Do Not Change!!!
```iecst
(** 2021-04-20 **)
PROGRAM _CYCLIC

	IF bInitialDone = FALSE THEN
		IF g_tyStartUp.bNtSettingsLoadDone = TRUE  THEN
			bInitialDone	:= TRUE;
			Act_Initial;
		END_IF

	ELSE

		Act_InputConfig;
		IF (tylocalDSSOT.In.bPrep = TRUE) AND (tylocalDSSOT.In.bEn = TRUE) AND (tylocalDSSOT.In.bDis = FALSE) THEN
			Act_Link;
			Act_Background;
			Act_Main;
		ELSE
			IF tylocalDSSOT.Out.eStat <> SOTActIdle THEN
				tylocalDSSOT.Out.eStatus	:= Done;
			ELSE
				tylocalDSSOT.Out.eStatus	:= Idle;
			END_IF
		END_IF
		Act_OutputConfig;
		Act_Alarm;

	END_IF

END_PROGRAM
```

#### Act_Link.st - Change By Project
```iecst
(** 3033-04-30 **)
ACTION Act_Link:

		//Ready Send
	tylocalDSSOT.In.bRdySend	:= TRUE;

	IF tylocalDSSOT.In.bLinkProjTCPAGVSigPrep THEN //TCP AGV
		tylocalDSSOT.In.bLeftSen := g_tyDInput.bOutMagConvExtSen;
		tylocalDSSOT.In.bRightSen := g_tyDInput.bOutMagConvMidSen;
		tylocalDSSOT.In.bDSB := g_tyTCP.bSvrDSB;

		//Send Complete Signal
		IF EDGENEG(tylocalDSSOT.In.bLeftSen) THEN
			tylocalDSSOT.In.bComplSigOn	:= TRUE;
		END_IF

		IF tylocalDSSOT.Out.eStat <> SOTActRun THEN
			tylocalDSSOT.In.bComplSigOn	:= FALSE;
		END_IF
	ELSE
		tylocalDSSOT.In.bLeftSen := g_tyDInput.bMagConvEntSen3;
		tylocalDSSOT.In.bRightSen := g_tyDInput.bMagPresentSen3;
		tylocalDSSOT.In.bDSB := g_tyDInput.bSOT3AIVReady;

		//Send Complete Signal
		IF EDGENEG(tylocalDSSOT.In.bLeftSen) THEN
			tylocalDSSOT.In.bComplSigOn	:= TRUE;
		END_IF

		IF tylocalDSSOT.Out.eStat <> SOTActRun THEN
			tylocalDSSOT.In.bComplSigOn	:= FALSE;
		END_IF

	END_IF

END_ACTION
```

#### Act_Alarm.st - Do Not Change!!!
```iecst
(** 2021-04-20 **)
ACTION Act_Alarm:
		//Reset Error
	IF (tylocalDSSOT.Out.eStatus = Error) AND bRstErr THEN
		tylocalDSSOT.In.eAct	:= MagConv2ClpActIdle;
		tylocalDSSOT.Out.eStat	:= MagConv2ClpActIdle;
	END_IF

	IF tylocalDSSOT.In.udiRstErr <> udiRstErrOld THEN
		bRstErr			:= TRUE;
		udiRstErrOld	:= tylocalDSSOT.In.udiRstErr;
	ELSE
		bRstErr			:= FALSE;
	END_IF
	//Error
	IF EDGEPOS(tylocalDSSOT.Out.eStatus = Error) THEN

		tylocalDSSOT.Out.tyAlmData.udiCode		:= udiStatus;
		tylocalDSSOT.Out.tyAlmData.eSeverity		:= AlmSeverityError;
		tylocalDSSOT.Out.tyAlmData.udiRunTime	:= tylocalDSSOT.Out.tyAlmData.udiRunTime + 1;
		tylocalDSSOT.Out.tyAlmData.bAlm			:= TRUE;
		tylocalDSSOT.Out.tyAlmData.udiModuleNum  := udiModuleNum;
		g_sDSSOTProgNm		    := tylocalDSSOT.In.sProgNm;

		tylocalDSSOT.Out.sStatTxt	:= tylocalDSSOT.Out.tyAlmData.sAlmMsg;

	ELSIF bRstErr AND (tyAlmData.udiCode <> 0) THEN

		tylocalDSSOT.Out.tyAlmData.udiCode	:= 0;
		tylocalDSSOT.Out.tyAlmData.eSeverity	:= AlmSeverityNA;
		tylocalDSSOT.Out.tyAlmData.bAlm			:= FALSE;
		tylocalDSSOT.Out.sStatTxt	:= a_sStatText[tylocalDSSOT.Out.eStat];

	END_IF

END_ACTION
```

#### Local.var - Do Not Change!!!
```iecst
(*2021-04-20*)
VAR
	tylocalDSSOT : tyDSSOT;
END_VAR
(**)
(*Local Action, State & Status*)
VAR
	eAct : eSOTAction;
	udiStatus : UDINT := 0;
	a_sStatText : ARRAY[0..50] OF STRING[200] := ['Idling','SMEMA Running','Turning On DBA Signal','Turning Off DBA Signal',47('')];
END_VAR
(**)
(**)
(*Local*)
VAR
	bRstErr : BOOL;
	udiRstErrOld : UDINT;
	bInitDone : BOOL;
	bInitialDone : BOOL;
	fbSOT : fbSOTDS;
	fbSigInChk : fbSOTSigInChk;
	eStatOld : eSOTAction := SOTActIdle;
	udiModuleNum : UDINT := 4501;
END_VAR
```

#### InputRef.var - not listed in the package file held
```iecst
(*2021-04-20*)
(**)
(*General*)
VAR
	p_eAct : REFERENCE TO eSOTAction;
	p_udiRstErr : REFERENCE TO UDINT;
	p_bPrep : REFERENCE TO BOOL;
	p_bEn : REFERENCE TO BOOL;
	p_bDis : REFERENCE TO BOOL;
END_VAR
(**)
(*Configuration*)
VAR
	p_bManual : REFERENCE TO BOOL;
	p_diTransferOutTO : REFERENCE TO DINT;
	p_bDirLToR : REFERENCE TO BOOL;
	p_bRdySend : REFERENCE TO BOOL;
END_VAR
(**)
(*Input*)
VAR
	p_bLeftSen : REFERENCE TO BOOL;
	p_bRightSen : REFERENCE TO BOOL;
	p_bComplSigOn : REFERENCE TO BOOL;
	p_bMagSizeLarge : REFERENCE TO BOOL;
	p_bDSB : REFERENCE TO BOOL;
	p_bVirtualEn : REFERENCE TO BOOL;
	p_bDSBVirtual : REFERENCE TO BOOL;
	p_tRstDlyTm : REFERENCE TO TIME;
	p_tSigInChkTm : REFERENCE TO TIME;
	p_sProgNm : REFERENCE TO STRING[15];
	p_bNtSettingsLoadDone : REFERENCE TO BOOL;
END_VAR
```

#### InputRef_Link.var - not listed in the package file held
```iecst
(*2021-04-20*)
(**)
VAR
	p_bLinkOpsRun : REFERENCE TO BOOL;
END_VAR
(**)
```

#### Act_Action.st - not listed in the package file held
```iecst
(** 2021-04-20 **)
ACTION Act_Action:

	//Reset Error
	IF (eStatus = Error) AND bRstErr THEN
		p_eAct	:= SOTActIdle;
		eStat	:= SOTActIdle;
	END_IF

	//Set p_eAct
	IF eStatus = Idle OR eStatus = Busy OR eStatus = Done THEN
		eStat	:= p_eAct;
	END_IF

END_ACTION
```

#### Act_InitGlobal.st - not listed in the package file held
```iecst
(** 2021-04-20 **)
ACTION Act_InitGlobal:

	(* Always Change If Project Change *)

	//Pass Data To Link
	p_bLinkOpsRun ACCESS p_OpsRun;

	//Pass Data To Internal Use
	p_udiRstErr ACCESS p_RstErrReset;
	p_bManual ACCESS p_UIMnlMod;
	p_diTransferOutTO ACCESS p_McParamTranInErrDlyTm;
	p_bEn ACCESS p_McParamAGVComEn;
//	p_bVirtualEn ACCESS p_UIVSOTDSEn;
//	p_bDSBVirtual ACCESS p_UIVSOTDSB;
	p_tRstDlyTm ACCESS p_NtParamDSSOT3RstDlyTm;
	p_tSigInChkTm ACCESS p_NtParamDSSOT3SigInChkTm;
	p_sProgNm ACCESS p_NtParamDSSOT3ProgNm;
	p_bNtSettingsLoadDone ACCESS p_StartupNtSettingsLoadDone;

	p_bMagSizeLarge ACCESS p_OpsMagConvUL3MagSizeL;

	(* Always Change If Project Change *)

END_ACTION
```

#### Act_LinkAction.st - not listed in the package file held
```iecst
(** 2021-04-20 **)
ACTION Act_LinkAction:

	IF p_bLinkOpsRun = TRUE THEN
		p_eAct ACCESS p_OpsMagConvUL3DSSOTAct;
	ELSE
		p_eAct ACCESS ADR(eAct);
	END_IF

END_ACTION
```

#### Act_RstErr.st - not listed in the package file held
```iecst
(** 2021-04-20 **)
ACTION Act_RstErr:

	IF p_udiRstErr <> udiRstErrOld THEN
		bRstErr			:= TRUE;
		udiRstErrOld	:= p_udiRstErr;
	ELSE
		bRstErr			:= FALSE;
	END_IF

END_ACTION
```

#### Init.st - not listed in the package file held
```iecst
(** 2021-04-20 **)
PROGRAM _INIT

	(* Always Change If Project Change *)

	//Pass Address To Global Address For External Use
	//Action, State & Status
	p_DSSOT3Stat		:= ADR(eStat);
	p_DSSOT3Status		:= ADR(eStatus);
	p_DSSOT3StatTxt		:= ADR(sStatTxt);

	//Alarm
	p_DSSOT3AlmData	:= ADR(tyAlmData);

	//Output
	p_DSSOT3USRdy			:= ADR(bUSRdy);
	p_DSSOT3DSRdy			:= ADR(bDSRdy);
	p_DSSOT3Transporting	:= ADR(bTransporting);
	p_DSSOT3ConvStart		:= ADR(bConvStart);
	p_DSSOT3ConvStop		:= ADR(bConvStop);
	p_DSSOT3DBA				:= ADR(bDBA);
	p_DSSOT3Virtual			:= ADR(bVirtual);
	p_DSSOT3MagSizeLarge	:= ADR(bDSMagSizeLarge);

	(* Always Change If Project Change *)

END_PROGRAM
```

### DSSOT1.var - not listed in the package file held
```iecst
(*2021-04-20*)
(**)
(*Action & State & Status*)
VAR
	p_DSSOT1Stat : UDINT;
	p_DSSOT1Status : UDINT;
	p_DSSOT1StatTxt : UDINT;
END_VAR
(**)
(*Alarm*)
VAR
	p_DSSOT1AlmData : UDINT;
END_VAR
(**)
(*Output*)
VAR
	p_DSSOT1USRdy : UDINT;
	p_DSSOT1DSRdy : UDINT;
	p_DSSOT1Transporting : UDINT;
	p_DSSOT1ConvStart : UDINT;
	p_DSSOT1ConvStop : UDINT;
	p_DSSOT1DBA : UDINT;
	p_DSSOT1MagSizeLarge : UDINT;
	p_DSSOT1Virtual : UDINT;
END_VAR
```

### DSSOT2.var - not listed in the package file held
```iecst
(*2021-04-20*)
(**)
(*Action & State & Status*)
VAR
	p_DSSOT2Stat : UDINT;
	p_DSSOT2Status : UDINT;
	p_DSSOT2StatTxt : UDINT;
END_VAR
(**)
(*Alarm*)
VAR
	p_DSSOT2AlmData : UDINT;
END_VAR
(**)
(*Output*)
VAR
	p_DSSOT2USRdy : UDINT;
	p_DSSOT2DSRdy : UDINT;
	p_DSSOT2Transporting : UDINT;
	p_DSSOT2ConvStart : UDINT;
	p_DSSOT2ConvStop : UDINT;
	p_DSSOT2DBA : UDINT;
	p_DSSOT2MagSizeLarge : UDINT;
	p_DSSOT2Virtual : UDINT;
END_VAR
```

### DSSOT3.var - not listed in the package file held
```iecst
(*2021-04-20*)
(**)
(*Action & State & Status*)
VAR
	p_DSSOT3Stat : UDINT;
	p_DSSOT3Status : UDINT;
	p_DSSOT3StatTxt : UDINT;
END_VAR
(**)
(*Alarm*)
VAR
	p_DSSOT3AlmData : UDINT;
END_VAR
(**)
(*Output*)
VAR
	p_DSSOT3USRdy : UDINT;
	p_DSSOT3DSRdy : UDINT;
	p_DSSOT3Transporting : UDINT;
	p_DSSOT3ConvStart : UDINT;
	p_DSSOT3ConvStop : UDINT;
	p_DSSOT3DBA : UDINT;
	p_DSSOT3MagSizeLarge : UDINT;
	p_DSSOT3Virtual : UDINT;
END_VAR
```

### USSOT1.var - not listed in the package file held
```iecst
(*2021-04-19*)
(**)
(*Action & State & Status*)
VAR
	p_USSOT1Stat : UDINT;
	p_USSOT1Status : UDINT;
	p_USSOT1StatTxt : UDINT;
END_VAR
(**)
(*Alarm*)
VAR
	p_USSOT1AlmData : UDINT;
END_VAR
(**)
(*Output*)
VAR
	p_USSOT1USRdy : UDINT;
	p_USSOT1USLargeMagRdy : UDINT;
	p_USSOT1DSRdy : UDINT;
	p_USSOT1Transporting : UDINT;
	p_USSOT1ConvStart : UDINT;
	p_USSOT1ConvStop : UDINT;
	p_USSOT1USB : UDINT;
	p_USSOT1Virtual : UDINT;
END_VAR
```

### USSOT2.var - not listed in the package file held
```iecst
(*2021-04-19*)
(**)
(*Action & State & Status*)
VAR
	p_USSOT2Stat : UDINT;
	p_USSOT2Status : UDINT;
	p_USSOT2StatTxt : UDINT;
END_VAR
(**)
(*Alarm*)
VAR
	p_USSOT2AlmData : UDINT;
END_VAR
(**)
(*Output*)
VAR
	p_USSOT2USRdy : UDINT;
	p_USSOT2USLargeMagRdy : UDINT;
	p_USSOT2DSRdy : UDINT;
	p_USSOT2Transporting : UDINT;
	p_USSOT2ConvStart : UDINT;
	p_USSOT2ConvStop : UDINT;
	p_USSOT2USB : UDINT;
	p_USSOT2Virtual : UDINT;
END_VAR
```

### USSOT3.var - not listed in the package file held
```iecst
(*2021-04-19*)
(**)
(*Action & State & Status*)
VAR
	p_USSOT3Stat : UDINT;
	p_USSOT3Status : UDINT;
	p_USSOT3StatTxt : UDINT;
END_VAR
(**)
(*Alarm*)
VAR
	p_USSOT3AlmData : UDINT;
END_VAR
(**)
(*Output*)
VAR
	p_USSOT3USRdy : UDINT;
	p_USSOT3USLargeMagRdy : UDINT;
	p_USSOT3DSRdy : UDINT;
	p_USSOT3Transporting : UDINT;
	p_USSOT3ConvStart : UDINT;
	p_USSOT3ConvStop : UDINT;
	p_USSOT3USB : UDINT;
	p_USSOT3Virtual : UDINT;
END_VAR
```
